(* Logix 5000 project; controller QW361 vendor 1 type 14 code 107 rev 32.11; software revision 32.00; part 17 of 20 *)

        [64].log_data[1].valid := 1, [64].log_data[2].time := 3599.999, [64].log_data[2].valid := 1, [64].log_data[3].time := 3599.999, [64].log_data[3].valid := 1, [64].log_data[4].min := 0.48812497, [64].log_data[4].max := 1.0068749, [64].log_data[4].total := 2935.025, [64].log_data[4].time := 3599.999, [64].log_data[4].minminute := 43, [64].log_data[4].maxminute := 34, [64].log_data[4].valid := 1, [64].log_data[5].max := 7.16125, [64].log_data[5].total := 3457.7583, [64].log_data[5].time := 3599.999, [64].log_data[5].maxminute := 35, [64].log_data[5].valid := 1, [64].log_data[6].valid := 1, [64].log_data[7].valid := 1, [64].log_data[8].valid := 1, [64].log_data[9].valid := 1, [64].log_data[10].valid := 1, [64].log_data[11].valid := 1, [64].log_data[12].valid := 1, [64].log_data[13].valid := 1, [64].log_data[14].valid := 1, [64].log_data[15].valid := 1, [64].log_data[16].valid := 1, [64].log_data[17].valid := 1, [64].log_data[18].valid := 1, [64].log_data[19].valid := 1, [64].time.Year := 2022, [64].time.Month := 4, [64].time.Day := 29, [64].time.Hour := 9, [64].time.Minute := 59, [64].time.Second := 59, [64].time.DST_ON := 1, [65].log_data[0].min := 1.0, [65].log_data[0].max := 1.0, [65].log_data[0].total := 3600.001, [65].log_data[0].time := 3600.001, [65].log_data[0].valid := 1, [65].log_data[1].time := 3600.001, [65].log_data[1].valid := 1, [65].log_data[2].max := 1.0, [65].log_data[2].total := 261.25, [65].log_data[2].time := 3600.001, [65].log_data[2].maxminute := 55, [65].log_data[2].valid := 1, [65].log_data[3].time := 3600.001, [65].log_data[3].valid := 1, [65].log_data[4].min := 0.64125, [65].log_data[4].max := 1.00875, [65].log_data[4].total := 3102.0618, [65].log_data[4].time := 3600.001, [65].log_data[4].maxminute := 55, [65].log_data[4].valid := 1, [65].log_data[5].max := 7.21375, [65].log_data[5].total := 1816.54,
        [65].log_data[5].time := 3600.001, [65].log_data[5].maxminute := 56, [65].log_data[5].valid := 1, [65].log_data[6].valid := 1, [65].log_data[7].valid := 1, [65].log_data[8].valid := 1, [65].log_data[9].valid := 1, [65].log_data[10].valid := 1, [65].log_data[11].valid := 1, [65].log_data[12].valid := 1, [65].log_data[13].valid := 1, [65].log_data[14].valid := 1, [65].log_data[15].valid := 1, [65].log_data[16].valid := 1, [65].log_data[17].valid := 1, [65].log_data[18].valid := 1, [65].log_data[19].valid := 1, [65].time.Year := 2022, [65].time.Month := 4, [65].time.Day := 29, [65].time.Hour := 10, [65].time.Minute := 59, [65].time.Second := 59, [65].time.DST_ON := 1, [66].log_data[0].min := 1.0, [66].log_data[0].max := 1.0, [66].log_data[0].total := 3600.0, [66].log_data[0].time := 3600.0, [66].log_data[0].valid := 1, [66].log_data[1].time := 3600.0, [66].log_data[1].valid := 1, [66].log_data[2].max := 1.0, [66].log_data[2].total := 236.25, [66].log_data[2].time := 3600.0, [66].log_data[2].minminute := 3, [66].log_data[2].valid := 1, [66].log_data[3].time := 3600.0, [66].log_data[3].valid := 1, [66].log_data[4].min := 0.48812497, [66].log_data[4].max := 0.93375, [66].log_data[4].total := 2553.6604, [66].log_data[4].time := 3600.0, [66].log_data[4].minminute := 4, [66].log_data[4].maxminute := 58, [66].log_data[4].valid := 1, [66].log_data[5].max := 7.1512504, [66].log_data[5].total := 1708.433, [66].log_data[5].time := 3600.0, [66].log_data[5].minminute := 4, [66].log_data[5].maxminute := 1, [66].log_data[5].valid := 1, [66].log_data[6].valid := 1, [66].log_data[7].valid := 1, [66].log_data[8].valid := 1, [66].log_data[9].valid := 1, [66].log_data[10].valid := 1, [66].log_data[11].valid := 1, [66].log_data[12].valid := 1, [66].log_data[13].valid := 1, [66].log_data[14].valid := 1,
        [66].log_data[15].valid := 1, [66].log_data[16].valid := 1, [66].log_data[17].valid := 1, [66].log_data[18].valid := 1, [66].log_data[19].valid := 1, [66].time.Year := 2022, [66].time.Month := 4, [66].time.Day := 29, [66].time.Hour := 11, [66].time.Minute := 59, [66].time.Second := 59, [66].time.DST_ON := 1, [67].log_data[0].min := 1.0, [67].log_data[0].max := 1.0, [67].log_data[0].total := 3600.0, [67].log_data[0].time := 3600.0, [67].log_data[0].valid := 1, [67].log_data[1].max := 1.0, [67].log_data[1].total := 497.5, [67].log_data[1].time := 3600.0, [67].log_data[1].maxminute := 16, [67].log_data[1].valid := 1, [67].log_data[2].time := 3600.0, [67].log_data[2].valid := 1, [67].log_data[3].time := 3600.0, [67].log_data[3].valid := 1, [67].log_data[4].min := 0.48812497, [67].log_data[4].max := 1.0024999, [67].log_data[4].total := 2646.7375, [67].log_data[4].time := 3600.0, [67].log_data[4].minminute := 24, [67].log_data[4].maxminute := 16, [67].log_data[4].valid := 1, [67].log_data[5].max := 7.1425004, [67].log_data[5].total := 3489.1882, [67].log_data[5].time := 3600.0, [67].log_data[5].maxminute := 17, [67].log_data[5].valid := 1, [67].log_data[6].valid := 1, [67].log_data[7].valid := 1, [67].log_data[8].valid := 1, [67].log_data[9].valid := 1, [67].log_data[10].valid := 1, [67].log_data[11].valid := 1, [67].log_data[12].valid := 1, [67].log_data[13].valid := 1, [67].log_data[14].valid := 1, [67].log_data[15].valid := 1, [67].log_data[16].valid := 1, [67].log_data[17].valid := 1, [67].log_data[18].valid := 1, [67].log_data[19].valid := 1, [67].time.Year := 2022, [67].time.Month := 4, [67].time.Day := 29, [67].time.Hour := 12, [67].time.Minute := 59, [67].time.Second := 59, [67].time.DST_ON := 1, [68].log_data[0].min := 1.0,
        [68].log_data[0].max := 1.0, [68].log_data[0].total := 3600.001, [68].log_data[0].time := 3600.001, [68].log_data[0].valid := 1, [68].log_data[1].time := 3600.001, [68].log_data[1].valid := 1, [68].log_data[2].time := 3600.001, [68].log_data[2].valid := 1, [68].log_data[3].time := 3600.001, [68].log_data[3].valid := 1, [68].log_data[4].min := 0.71812505, [68].log_data[4].max := 0.94875, [68].log_data[4].total := 3074.6538, [68].log_data[4].time := 3600.001, [68].log_data[4].maxminute := 56, [68].log_data[4].valid := 1, [68].log_data[5].time := 3600.001, [68].log_data[5].valid := 1, [68].log_data[6].valid := 1, [68].log_data[7].valid := 1, [68].log_data[8].valid := 1, [68].log_data[9].valid := 1, [68].log_data[10].valid := 1, [68].log_data[11].valid := 1, [68].log_data[12].valid := 1, [68].log_data[13].valid := 1, [68].log_data[14].valid := 1, [68].log_data[15].valid := 1, [68].log_data[16].valid := 1, [68].log_data[17].valid := 1, [68].log_data[18].valid := 1, [68].log_data[19].valid := 1, [68].time.Year := 2022, [68].time.Month := 4, [68].time.Day := 29, [68].time.Hour := 13, [68].time.Minute := 59, [68].time.Second := 59, [68].time.DST_ON := 1, [69].log_data[0].min := 1.0, [69].log_data[0].max := 1.0, [69].log_data[0].total := 3599.999, [69].log_data[0].time := 3599.999, [69].log_data[0].valid := 1, [69].log_data[1].time := 3599.999, [69].log_data[1].valid := 1, [69].log_data[2].max := 1.0, [69].log_data[2].total := 480.5, [69].log_data[2].time := 3599.999, [69].log_data[2].maxminute := 26, [69].log_data[2].valid := 1, [69].log_data[3].time := 3599.999, [69].log_data[3].valid := 1, [69].log_data[4].min := 0.48749998, [69].log_data[4].max := 1.0068749, [69].log_data[4].total := 2784.5537, [69].log_data[4].time := 3599.999, [69].log_data[4].minminute := 34, [69].log_data[4].maxminute := 26, [69].log_data[4].valid := 1,
        [69].log_data[5].max := 7.2375, [69].log_data[5].total := 3409.78, [69].log_data[5].time := 3599.999, [69].log_data[5].maxminute := 26, [69].log_data[5].valid := 1, [69].log_data[6].valid := 1, [69].log_data[7].valid := 1, [69].log_data[8].valid := 1, [69].log_data[9].valid := 1, [69].log_data[10].valid := 1, [69].log_data[11].valid := 1, [69].log_data[12].valid := 1, [69].log_data[13].valid := 1, [69].log_data[14].valid := 1, [69].log_data[15].valid := 1, [69].log_data[16].valid := 1, [69].log_data[17].valid := 1, [69].log_data[18].valid := 1, [69].log_data[19].valid := 1, [69].time.Year := 2022, [69].time.Month := 4, [69].time.Day := 29, [69].time.Hour := 14, [69].time.Minute := 59, [69].time.Second := 59, [69].time.DST_ON := 1, [70].log_data[0].min := 1.0, [70].log_data[0].max := 1.0, [70].log_data[0].total := 3600.001, [70].log_data[0].time := 3600.001, [70].log_data[0].valid := 1, [70].log_data[1].time := 3600.001, [70].log_data[1].valid := 1, [70].log_data[2].time := 3600.001, [70].log_data[2].valid := 1, [70].log_data[3].time := 3600.001, [70].log_data[3].valid := 1, [70].log_data[4].min := 0.64187497, [70].log_data[4].max := 0.91875005, [70].log_data[4].total := 2832.5027, [70].log_data[4].time := 3600.001, [70].log_data[4].maxminute := 56, [70].log_data[4].valid := 1, [70].log_data[5].time := 3600.001, [70].log_data[5].valid := 1, [70].log_data[6].valid := 1, [70].log_data[7].valid := 1, [70].log_data[8].valid := 1, [70].log_data[9].valid := 1, [70].log_data[10].valid := 1, [70].log_data[11].valid := 1, [70].log_data[12].valid := 1, [70].log_data[13].valid := 1, [70].log_data[14].valid := 1, [70].log_data[15].valid := 1, [70].log_data[16].valid := 1, [70].log_data[17].valid := 1, [70].log_data[18].valid := 1, [70].log_data[19].valid := 1, [70].time.Year := 2022,
        [70].time.Month := 4, [70].time.Day := 29, [70].time.Hour := 15, [70].time.Minute := 59, [70].time.Second := 59, [70].time.DST_ON := 1, [71].log_data[0].min := 1.0, [71].log_data[0].max := 1.0, [71].log_data[0].total := 3600.0, [71].log_data[0].time := 3600.0, [71].log_data[0].valid := 1, [71].log_data[1].max := 1.0, [71].log_data[1].total := 486.0, [71].log_data[1].time := 3600.0, [71].log_data[1].maxminute := 33, [71].log_data[1].valid := 1, [71].log_data[2].time := 3600.0, [71].log_data[2].valid := 1, [71].log_data[3].time := 3600.0, [71].log_data[3].valid := 1, [71].log_data[4].min := 0.48749998, [71].log_data[4].max := 1.00375, [71].log_data[4].total := 2909.2458, [71].log_data[4].time := 3600.0, [71].log_data[4].minminute := 41, [71].log_data[4].maxminute := 33, [71].log_data[4].valid := 1, [71].log_data[5].max := 7.1525, [71].log_data[5].total := 3410.604, [71].log_data[5].time := 3600.0, [71].log_data[5].maxminute := 34, [71].log_data[5].valid := 1, [71].log_data[6].valid := 1, [71].log_data[7].valid := 1, [71].log_data[8].valid := 1, [71].log_data[9].valid := 1, [71].log_data[10].valid := 1, [71].log_data[11].valid := 1, [71].log_data[12].valid := 1, [71].log_data[13].valid := 1, [71].log_data[14].valid := 1, [71].log_data[15].valid := 1, [71].log_data[16].valid := 1, [71].log_data[17].valid := 1, [71].log_data[18].valid := 1, [71].log_data[19].valid := 1, [71].time.Year := 2022, [71].time.Month := 4, [71].time.Day := 29, [71].time.Hour := 16, [71].time.Minute := 59, [71].time.Second := 59, [71].time.DST_ON := 1, [72].log_data[0].min := 1.0, [72].log_data[0].max := 1.0, [72].log_data[0].total := 3599.999, [72].log_data[0].time := 3599.999, [72].log_data[0].valid := 1, [72].log_data[1].time := 3599.999, [72].log_data[1].valid := 1,
        [72].log_data[2].time := 3599.999, [72].log_data[2].valid := 1, [72].log_data[3].time := 3599.999, [72].log_data[3].valid := 1, [72].log_data[4].min := 0.57937497, [72].log_data[4].max := 0.8725, [72].log_data[4].total := 2595.1763, [72].log_data[4].time := 3599.999, [72].log_data[4].maxminute := 59, [72].log_data[4].valid := 1, [72].log_data[5].time := 3599.999, [72].log_data[5].valid := 1, [72].log_data[6].valid := 1, [72].log_data[7].valid := 1, [72].log_data[8].valid := 1, [72].log_data[9].valid := 1, [72].log_data[10].valid := 1, [72].log_data[11].valid := 1, [72].log_data[12].valid := 1, [72].log_data[13].valid := 1, [72].log_data[14].valid := 1, [72].log_data[15].valid := 1, [72].log_data[16].valid := 1, [72].log_data[17].valid := 1, [72].log_data[18].valid := 1, [72].log_data[19].valid := 1, [72].time.Year := 2022, [72].time.Month := 4, [72].time.Day := 29, [72].time.Hour := 17, [72].time.Minute := 59, [72].time.Second := 59, [72].time.DST_ON := 1, [73].log_data[0].min := 1.0, [73].log_data[0].max := 1.0, [73].log_data[0].total := 3600.0, [73].log_data[0].time := 3600.0, [73].log_data[0].valid := 1, [73].log_data[1].time := 3600.0, [73].log_data[1].valid := 1, [73].log_data[2].max := 1.0, [73].log_data[2].total := 486.0, [73].log_data[2].time := 3600.0, [73].log_data[2].maxminute := 50, [73].log_data[2].valid := 1, [73].log_data[3].time := 3600.0, [73].log_data[3].valid := 1, [73].log_data[4].min := 0.48749998, [73].log_data[4].max := 1.00625, [73].log_data[4].total := 3274.2031, [73].log_data[4].time := 3600.0, [73].log_data[4].minminute := 58, [73].log_data[4].maxminute := 50, [73].log_data[4].valid := 1, [73].log_data[5].max := 7.235, [73].log_data[5].total := 3447.0845, [73].log_data[5].time := 3600.0, [73].log_data[5].maxminute := 51, [73].log_data[5].valid := 1, [73].log_data[6].valid := 1,
        [73].log_data[7].valid := 1, [73].log_data[8].valid := 1, [73].log_data[9].valid := 1, [73].log_data[10].valid := 1, [73].log_data[11].valid := 1, [73].log_data[12].valid := 1, [73].log_data[13].valid := 1, [73].log_data[14].valid := 1, [73].log_data[15].valid := 1, [73].log_data[16].valid := 1, [73].log_data[17].valid := 1, [73].log_data[18].valid := 1, [73].log_data[19].valid := 1, [73].time.Year := 2022, [73].time.Month := 4, [73].time.Day := 29, [73].time.Hour := 18, [73].time.Minute := 59, [73].time.Second := 59, [73].time.DST_ON := 1, [74].log_data[0].min := 1.0, [74].log_data[0].max := 1.0, [74].log_data[0].total := 3600.0, [74].log_data[0].time := 3600.0, [74].log_data[0].valid := 1, [74].log_data[1].time := 3600.0, [74].log_data[1].valid := 1, [74].log_data[2].time := 3600.0, [74].log_data[2].valid := 1, [74].log_data[3].time := 3600.0, [74].log_data[3].valid := 1, [74].log_data[4].min := 0.48749998, [74].log_data[4].max := 0.9024999, [74].log_data[4].total := 2510.1887, [74].log_data[4].time := 3600.0, [74].log_data[4].maxminute := 57, [74].log_data[4].valid := 1, [74].log_data[5].time := 3600.0, [74].log_data[5].valid := 1, [74].log_data[6].valid := 1, [74].log_data[7].valid := 1, [74].log_data[8].valid := 1, [74].log_data[9].valid := 1, [74].log_data[10].valid := 1, [74].log_data[11].valid := 1, [74].log_data[12].valid := 1, [74].log_data[13].valid := 1, [74].log_data[14].valid := 1, [74].log_data[15].valid := 1, [74].log_data[16].valid := 1, [74].log_data[17].valid := 1, [74].log_data[18].valid := 1, [74].log_data[19].valid := 1, [74].time.Year := 2022, [74].time.Month := 4, [74].time.Day := 29, [74].time.Hour := 19, [74].time.Minute := 59, [74].time.Second := 59, [74].time.DST_ON := 1,
        [75].log_data[0].min := 1.0, [75].log_data[0].max := 1.0, [75].log_data[0].total := 3599.999, [75].log_data[0].time := 3599.999, [75].log_data[0].valid := 1, [75].log_data[1].max := 1.0, [75].log_data[1].total := 512.0, [75].log_data[1].time := 3599.999, [75].log_data[1].maxminute := 25, [75].log_data[1].valid := 1, [75].log_data[2].time := 3599.999, [75].log_data[2].valid := 1, [75].log_data[3].time := 3599.999, [75].log_data[3].valid := 1, [75].log_data[4].min := 0.48749998, [75].log_data[4].max := 1.00875, [75].log_data[4].total := 2836.993, [75].log_data[4].time := 3599.999, [75].log_data[4].minminute := 34, [75].log_data[4].maxminute := 25, [75].log_data[4].valid := 1, [75].log_data[5].max := 7.1650004, [75].log_data[5].total := 3593.2307, [75].log_data[5].time := 3599.999, [75].log_data[5].maxminute := 26, [75].log_data[5].valid := 1, [75].log_data[6].valid := 1, [75].log_data[7].valid := 1, [75].log_data[8].valid := 1, [75].log_data[9].valid := 1, [75].log_data[10].valid := 1, [75].log_data[11].valid := 1, [75].log_data[12].valid := 1, [75].log_data[13].valid := 1, [75].log_data[14].valid := 1, [75].log_data[15].valid := 1, [75].log_data[16].valid := 1, [75].log_data[17].valid := 1, [75].log_data[18].valid := 1, [75].log_data[19].valid := 1, [75].time.Year := 2022, [75].time.Month := 4, [75].time.Day := 29, [75].time.Hour := 20, [75].time.Minute := 59, [75].time.Second := 59, [75].time.DST_ON := 1, [76].log_data[0].min := 1.0, [76].log_data[0].max := 1.0, [76].log_data[0].total := 3600.0, [76].log_data[0].time := 3600.0, [76].log_data[0].valid := 1, [76].log_data[1].time := 3600.0, [76].log_data[1].valid := 1, [76].log_data[2].max := 1.0, [76].log_data[2].total := 493.0, [76].log_data[2].time := 3600.0, [76].log_data[2].maxminute := 50, [76].log_data[2].valid := 1, [76].log_data[3].time := 3600.0,
        [76].log_data[3].valid := 1, [76].log_data[4].min := 0.48812497, [76].log_data[4].max := 1.005, [76].log_data[4].total := 3163.5645, [76].log_data[4].time := 3600.0, [76].log_data[4].minminute := 58, [76].log_data[4].maxminute := 50, [76].log_data[4].valid := 1, [76].log_data[5].max := 7.24375, [76].log_data[5].total := 3493.379, [76].log_data[5].time := 3600.0, [76].log_data[5].maxminute := 50, [76].log_data[5].valid := 1, [76].log_data[6].valid := 1, [76].log_data[7].valid := 1, [76].log_data[8].valid := 1, [76].log_data[9].valid := 1, [76].log_data[10].valid := 1, [76].log_data[11].valid := 1, [76].log_data[12].valid := 1, [76].log_data[13].valid := 1, [76].log_data[14].valid := 1, [76].log_data[15].valid := 1, [76].log_data[16].valid := 1, [76].log_data[17].valid := 1, [76].log_data[18].valid := 1, [76].log_data[19].valid := 1, [76].time.Year := 2022, [76].time.Month := 4, [76].time.Day := 29, [76].time.Hour := 21, [76].time.Minute := 59, [76].time.Second := 59, [76].time.DST_ON := 1, [77].log_data[0].min := 1.0, [77].log_data[0].max := 1.0, [77].log_data[0].total := 3600.0, [77].log_data[0].time := 3600.0, [77].log_data[0].valid := 1, [77].log_data[1].time := 3600.0, [77].log_data[1].valid := 1, [77].log_data[2].time := 3600.0, [77].log_data[2].valid := 1, [77].log_data[3].time := 3600.0, [77].log_data[3].valid := 1, [77].log_data[4].min := 0.5025, [77].log_data[4].max := 0.94875, [77].log_data[4].total := 2784.093, [77].log_data[4].time := 3600.0, [77].log_data[4].maxminute := 57, [77].log_data[4].valid := 1, [77].log_data[5].max := 0.0025000002, [77].log_data[5].total := 0.59032303, [77].log_data[5].time := 3600.0, [77].log_data[5].maxminute := 54, [77].log_data[5].valid := 1, [77].log_data[6].valid := 1, [77].log_data[7].valid := 1, [77].log_data[8].valid := 1, [77].log_data[9].valid := 1,
        [77].log_data[10].valid := 1, [77].log_data[11].valid := 1, [77].log_data[12].valid := 1, [77].log_data[13].valid := 1, [77].log_data[14].valid := 1, [77].log_data[15].valid := 1, [77].log_data[16].valid := 1, [77].log_data[17].valid := 1, [77].log_data[18].valid := 1, [77].log_data[19].valid := 1, [77].time.Year := 2022, [77].time.Month := 4, [77].time.Day := 29, [77].time.Hour := 22, [77].time.Minute := 59, [77].time.Second := 59, [77].time.DST_ON := 1, [78].log_data[0].min := 1.0, [78].log_data[0].max := 1.0, [78].log_data[0].total := 3600.0, [78].log_data[0].time := 3600.0, [78].log_data[0].valid := 1, [78].log_data[1].max := 1.0, [78].log_data[1].total := 483.5, [78].log_data[1].time := 3600.0, [78].log_data[1].maxminute := 24, [78].log_data[1].valid := 1, [78].log_data[2].time := 3600.0, [78].log_data[2].valid := 1, [78].log_data[3].time := 3600.0, [78].log_data[3].valid := 1, [78].log_data[4].min := 0.48812497, [78].log_data[4].max := 1.0068749, [78].log_data[4].total := 2779.4797, [78].log_data[4].time := 3600.0, [78].log_data[4].minminute := 32, [78].log_data[4].maxminute := 24, [78].log_data[4].valid := 1, [78].log_data[5].max := 7.13875, [78].log_data[5].total := 3404.901, [78].log_data[5].time := 3600.0, [78].log_data[5].maxminute := 25, [78].log_data[5].valid := 1, [78].log_data[6].valid := 1, [78].log_data[7].valid := 1, [78].log_data[8].valid := 1, [78].log_data[9].valid := 1, [78].log_data[10].valid := 1, [78].log_data[11].valid := 1, [78].log_data[12].valid := 1, [78].log_data[13].valid := 1, [78].log_data[14].valid := 1, [78].log_data[15].valid := 1, [78].log_data[16].valid := 1, [78].log_data[17].valid := 1, [78].log_data[18].valid := 1, [78].log_data[19].valid := 1, [78].time.Year := 2022, [78].time.Month := 4, [78].time.Day := 29,
        [78].time.Hour := 23, [78].time.Minute := 59, [78].time.Second := 59, [78].time.DST_ON := 1, [79].log_data[0].min := 1.0, [79].log_data[0].max := 1.0, [79].log_data[0].total := 3600.0, [79].log_data[0].time := 3600.0, [79].log_data[0].valid := 1, [79].log_data[1].time := 3600.0, [79].log_data[1].valid := 1, [79].log_data[2].time := 3600.0, [79].log_data[2].valid := 1, [79].log_data[3].time := 3600.0, [79].log_data[3].valid := 1, [79].log_data[4].min := 0.71812505, [79].log_data[4].max := 0.98, [79].log_data[4].total := 3211.9824, [79].log_data[4].time := 3600.0, [79].log_data[4].maxminute := 53, [79].log_data[4].valid := 1, [79].log_data[5].max := 0.0012500001, [79].log_data[5].total := 1.0756322, [79].log_data[5].time := 3600.0, [79].log_data[5].valid := 1, [79].log_data[6].valid := 1, [79].log_data[7].valid := 1, [79].log_data[8].valid := 1, [79].log_data[9].valid := 1, [79].log_data[10].valid := 1, [79].log_data[11].valid := 1, [79].log_data[12].valid := 1, [79].log_data[13].valid := 1, [79].log_data[14].valid := 1, [79].log_data[15].valid := 1, [79].log_data[16].valid := 1, [79].log_data[17].valid := 1, [79].log_data[18].valid := 1, [79].log_data[19].valid := 1, [79].time.Year := 2022, [79].time.Month := 4, [79].time.Day := 30, [79].time.Minute := 59, [79].time.Second := 59, [79].time.DST_ON := 1, [80].log_data[0].min := 1.0, [80].log_data[0].max := 1.0, [80].log_data[0].total := 3600.0, [80].log_data[0].time := 3600.0, [80].log_data[0].valid := 1, [80].log_data[1].time := 3600.0, [80].log_data[1].valid := 1, [80].log_data[2].max := 1.0, [80].log_data[2].total := 477.0, [80].log_data[2].time := 3600.0, [80].log_data[2].maxminute := 10, [80].log_data[2].valid := 1, [80].log_data[3].time := 3600.0, [80].log_data[3].valid := 1, [80].log_data[4].min := 0.48812497,
        [80].log_data[4].max := 1.0068749, [80].log_data[4].total := 2421.8188, [80].log_data[4].time := 3600.0, [80].log_data[4].minminute := 18, [80].log_data[4].maxminute := 10, [80].log_data[4].valid := 1, [80].log_data[5].max := 7.2237496, [80].log_data[5].total := 3382.9375, [80].log_data[5].time := 3600.0, [80].log_data[5].maxminute := 11, [80].log_data[5].valid := 1, [80].log_data[6].valid := 1, [80].log_data[7].valid := 1, [80].log_data[8].valid := 1, [80].log_data[9].valid := 1, [80].log_data[10].valid := 1, [80].log_data[11].valid := 1, [80].log_data[12].valid := 1, [80].log_data[13].valid := 1, [80].log_data[14].valid := 1, [80].log_data[15].valid := 1, [80].log_data[16].valid := 1, [80].log_data[17].valid := 1, [80].log_data[18].valid := 1, [80].log_data[19].valid := 1, [80].time.Year := 2022, [80].time.Month := 4, [80].time.Day := 30, [80].time.Hour := 1, [80].time.Minute := 59, [80].time.Second := 59, [80].time.DST_ON := 1, [81].log_data[0].min := 1.0, [81].log_data[0].max := 1.0, [81].log_data[0].total := 3600.0, [81].log_data[0].time := 3600.0, [81].log_data[0].valid := 1, [81].log_data[1].time := 3600.0, [81].log_data[1].valid := 1, [81].log_data[2].time := 3600.0, [81].log_data[2].valid := 1, [81].log_data[3].time := 3600.0, [81].log_data[3].valid := 1, [81].log_data[4].min := 0.656875, [81].log_data[4].max := 0.8268749, [81].log_data[4].total := 2698.259, [81].log_data[4].time := 3600.0, [81].log_data[4].maxminute := 55, [81].log_data[4].valid := 1, [81].log_data[5].max := 0.0012500001, [81].log_data[5].total := 2.276786, [81].log_data[5].time := 3600.0, [81].log_data[5].valid := 1, [81].log_data[6].valid := 1, [81].log_data[7].valid := 1, [81].log_data[8].valid := 1, [81].log_data[9].valid := 1, [81].log_data[10].valid := 1, [81].log_data[11].valid := 1, [81].log_data[12].valid := 1,
        [81].log_data[13].valid := 1, [81].log_data[14].valid := 1, [81].log_data[15].valid := 1, [81].log_data[16].valid := 1, [81].log_data[17].valid := 1, [81].log_data[18].valid := 1, [81].log_data[19].valid := 1, [81].time.Year := 2022, [81].time.Month := 4, [81].time.Day := 30, [81].time.Hour := 2, [81].time.Minute := 59, [81].time.Second := 59, [81].time.DST_ON := 1, [82].log_data[0].min := 1.0, [82].log_data[0].max := 1.0, [82].log_data[0].total := 3600.0, [82].log_data[0].time := 3600.0, [82].log_data[0].valid := 1, [82].log_data[1].time := 3600.0, [82].log_data[1].valid := 1, [82].log_data[2].time := 3600.0, [82].log_data[2].valid := 1, [82].log_data[3].time := 3600.0, [82].log_data[3].valid := 1, [82].log_data[4].min := 0.82625, [82].log_data[4].max := 0.91875005, [82].log_data[4].total := 3186.939, [82].log_data[4].time := 3600.0, [82].log_data[4].maxminute := 48, [82].log_data[4].valid := 1, [82].log_data[5].max := 0.0012500001, [82].log_data[5].total := 2.8984814, [82].log_data[5].time := 3600.0, [82].log_data[5].valid := 1, [82].log_data[6].valid := 1, [82].log_data[7].valid := 1, [82].log_data[8].valid := 1, [82].log_data[9].valid := 1, [82].log_data[10].valid := 1, [82].log_data[11].valid := 1, [82].log_data[12].valid := 1, [82].log_data[13].valid := 1, [82].log_data[14].valid := 1, [82].log_data[15].valid := 1, [82].log_data[16].valid := 1, [82].log_data[17].valid := 1, [82].log_data[18].valid := 1, [82].log_data[19].valid := 1, [82].time.Year := 2022, [82].time.Month := 4, [82].time.Day := 30, [82].time.Hour := 3, [82].time.Minute := 59, [82].time.Second := 59, [82].time.DST_ON := 1, [83].log_data[0].min := 1.0, [83].log_data[0].max := 1.0, [83].log_data[0].total := 3600.0, [83].log_data[0].time := 3600.0,
        [83].log_data[0].valid := 1, [83].log_data[1].time := 3600.0, [83].log_data[1].valid := 1, [83].log_data[2].time := 3600.0, [83].log_data[2].valid := 1, [83].log_data[3].time := 3600.0, [83].log_data[3].valid := 1, [83].log_data[4].min := 0.91875005, [83].log_data[4].max := 0.9650001, [83].log_data[4].total := 3411.9158, [83].log_data[4].time := 3600.0, [83].log_data[4].maxminute := 42, [83].log_data[4].valid := 1, [83].log_data[5].max := 0.0012500001, [83].log_data[5].total := 2.8228402, [83].log_data[5].time := 3600.0, [83].log_data[5].valid := 1, [83].log_data[6].valid := 1, [83].log_data[7].valid := 1, [83].log_data[8].valid := 1, [83].log_data[9].valid := 1, [83].log_data[10].valid := 1, [83].log_data[11].valid := 1, [83].log_data[12].valid := 1, [83].log_data[13].valid := 1, [83].log_data[14].valid := 1, [83].log_data[15].valid := 1, [83].log_data[16].valid := 1, [83].log_data[17].valid := 1, [83].log_data[18].valid := 1, [83].log_data[19].valid := 1, [83].time.Year := 2022, [83].time.Month := 4, [83].time.Day := 30, [83].time.Hour := 4, [83].time.Minute := 59, [83].time.Second := 59, [83].time.DST_ON := 1, [84].log_data[0].min := 1.0, [84].log_data[0].max := 1.0, [84].log_data[0].total := 3599.999, [84].log_data[0].time := 3599.999, [84].log_data[0].valid := 1, [84].log_data[1].max := 1.0, [84].log_data[1].total := 154.75, [84].log_data[1].time := 3599.999, [84].log_data[1].maxminute := 57, [84].log_data[1].valid := 1, [84].log_data[2].time := 3599.999, [84].log_data[2].valid := 1, [84].log_data[3].time := 3599.999, [84].log_data[3].valid := 1, [84].log_data[4].min := 0.9125, [84].log_data[4].max := 1.00125, [84].log_data[4].total := 3550.91, [84].log_data[4].time := 3599.999, [84].log_data[4].minminute := 59, [84].log_data[4].maxminute := 57, [84].log_data[4].valid := 1, [84].log_data[5].max := 7.1625,
        [84].log_data[5].total := 1047.2858, [84].log_data[5].time := 3599.999, [84].log_data[5].maxminute := 58, [84].log_data[5].valid := 1, [84].log_data[6].valid := 1, [84].log_data[7].valid := 1, [84].log_data[8].valid := 1, [84].log_data[9].valid := 1, [84].log_data[10].valid := 1, [84].log_data[11].valid := 1, [84].log_data[12].valid := 1, [84].log_data[13].valid := 1, [84].log_data[14].valid := 1, [84].log_data[15].valid := 1, [84].log_data[16].valid := 1, [84].log_data[17].valid := 1, [84].log_data[18].valid := 1, [84].log_data[19].valid := 1, [84].time.Year := 2022, [84].time.Month := 4, [84].time.Day := 30, [84].time.Hour := 5, [84].time.Minute := 59, [84].time.Second := 59, [84].time.DST_ON := 1, [85].log_data[0].min := 1.0, [85].log_data[0].max := 1.0, [85].log_data[0].total := 3600.0, [85].log_data[0].time := 3600.0, [85].log_data[0].valid := 1, [85].log_data[1].max := 1.0, [85].log_data[1].total := 317.25, [85].log_data[1].time := 3600.0, [85].log_data[1].minminute := 5, [85].log_data[1].valid := 1, [85].log_data[2].time := 3600.0, [85].log_data[2].valid := 1, [85].log_data[3].time := 3600.0, [85].log_data[3].valid := 1, [85].log_data[4].min := 0.48812497, [85].log_data[4].max := 0.9125, [85].log_data[4].total := 1935.4558, [85].log_data[4].time := 3600.0, [85].log_data[4].minminute := 5, [85].log_data[4].valid := 1, [85].log_data[5].max := 7.1225, [85].log_data[5].total := 2269.2898, [85].log_data[5].time := 3600.0, [85].log_data[5].minminute := 5, [85].log_data[5].valid := 1, [85].log_data[6].valid := 1, [85].log_data[7].valid := 1, [85].log_data[8].valid := 1, [85].log_data[9].valid := 1, [85].log_data[10].valid := 1, [85].log_data[11].valid := 1, [85].log_data[12].valid := 1, [85].log_data[13].valid := 1, [85].log_data[14].valid := 1, [85].log_data[15].valid := 1,
        [85].log_data[16].valid := 1, [85].log_data[17].valid := 1, [85].log_data[18].valid := 1, [85].log_data[19].valid := 1, [85].time.Year := 2022, [85].time.Month := 4, [85].time.Day := 30, [85].time.Hour := 6, [85].time.Minute := 59, [85].time.Second := 59, [85].time.DST_ON := 1, [86].log_data[0].min := 1.0, [86].log_data[0].max := 1.0, [86].log_data[0].total := 3600.0, [86].log_data[0].time := 3600.0, [86].log_data[0].valid := 1, [86].log_data[1].time := 3600.0, [86].log_data[1].valid := 1, [86].log_data[2].time := 3600.0, [86].log_data[2].valid := 1, [86].log_data[3].time := 3600.0, [86].log_data[3].valid := 1, [86].log_data[4].min := 0.56500006, [86].log_data[4].max := 0.70375, [86].log_data[4].total := 2291.6409, [86].log_data[4].time := 3600.0, [86].log_data[4].maxminute := 55, [86].log_data[4].valid := 1, [86].log_data[5].max := 0.0025000002, [86].log_data[5].total := 1.7577057, [86].log_data[5].time := 3600.0, [86].log_data[5].maxminute := 35, [86].log_data[5].valid := 1, [86].log_data[6].valid := 1, [86].log_data[7].valid := 1, [86].log_data[8].valid := 1, [86].log_data[9].valid := 1, [86].log_data[10].valid := 1, [86].log_data[11].valid := 1, [86].log_data[12].valid := 1, [86].log_data[13].valid := 1, [86].log_data[14].valid := 1, [86].log_data[15].valid := 1, [86].log_data[16].valid := 1, [86].log_data[17].valid := 1, [86].log_data[18].valid := 1, [86].log_data[19].valid := 1, [86].time.Year := 2022, [86].time.Month := 4, [86].time.Day := 30, [86].time.Hour := 7, [86].time.Minute := 59, [86].time.Second := 59, [86].time.DST_ON := 1, [87].log_data[0].min := 1.0, [87].log_data[0].max := 1.0, [87].log_data[0].total := 3599.999, [87].log_data[0].time := 3599.999, [87].log_data[0].valid := 1, [87].log_data[1].time := 3599.999,
        [87].log_data[1].valid := 1, [87].log_data[2].time := 3599.999, [87].log_data[2].valid := 1, [87].log_data[3].time := 3599.999, [87].log_data[3].valid := 1, [87].log_data[4].min := 0.703125, [87].log_data[4].max := 0.9024999, [87].log_data[4].total := 2915.0146, [87].log_data[4].time := 3599.999, [87].log_data[4].maxminute := 55, [87].log_data[4].valid := 1, [87].log_data[5].max := 0.0025000002, [87].log_data[5].total := 0.7278249, [87].log_data[5].time := 3599.999, [87].log_data[5].maxminute := 1, [87].log_data[5].valid := 1, [87].log_data[6].valid := 1, [87].log_data[7].valid := 1, [87].log_data[8].valid := 1, [87].log_data[9].valid := 1, [87].log_data[10].valid := 1, [87].log_data[11].valid := 1, [87].log_data[12].valid := 1, [87].log_data[13].valid := 1, [87].log_data[14].valid := 1, [87].log_data[15].valid := 1, [87].log_data[16].valid := 1, [87].log_data[17].valid := 1, [87].log_data[18].valid := 1, [87].log_data[19].valid := 1, [87].time.Year := 2022, [87].time.Month := 4, [87].time.Day := 30, [87].time.Hour := 8, [87].time.Minute := 59, [87].time.Second := 59, [87].time.DST_ON := 1, [88].log_data[0].min := 1.0, [88].log_data[0].max := 1.0, [88].log_data[0].total := 3600.0, [88].log_data[0].time := 3600.0, [88].log_data[0].valid := 1, [88].log_data[1].time := 3600.0, [88].log_data[1].valid := 1, [88].log_data[2].max := 1.0, [88].log_data[2].total := 527.0, [88].log_data[2].time := 3600.0, [88].log_data[2].maxminute := 24, [88].log_data[2].valid := 1, [88].log_data[3].time := 3600.0, [88].log_data[3].valid := 1, [88].log_data[4].min := 0.48812497, [88].log_data[4].max := 1.00875, [88].log_data[4].total := 2933.3132, [88].log_data[4].time := 3600.0, [88].log_data[4].minminute := 33, [88].log_data[4].maxminute := 24, [88].log_data[4].valid := 1, [88].log_data[5].max := 7.2199993, [88].log_data[5].total := 3743.0854,
        [88].log_data[5].time := 3600.0, [88].log_data[5].maxminute := 25, [88].log_data[5].valid := 1, [88].log_data[6].valid := 1, [88].log_data[7].valid := 1, [88].log_data[8].valid := 1, [88].log_data[9].valid := 1, [88].log_data[10].valid := 1, [88].log_data[11].valid := 1, [88].log_data[12].valid := 1, [88].log_data[13].valid := 1, [88].log_data[14].valid := 1, [88].log_data[15].valid := 1, [88].log_data[16].valid := 1, [88].log_data[17].valid := 1, [88].log_data[18].valid := 1, [88].log_data[19].valid := 1, [88].time.Year := 2022, [88].time.Month := 4, [88].time.Day := 30, [88].time.Hour := 9, [88].time.Minute := 59, [88].time.Second := 59, [88].time.DST_ON := 1, [89].log_data[0].min := 1.0, [89].log_data[0].max := 1.0, [89].log_data[0].total := 3600.0, [89].log_data[0].time := 3600.0, [89].log_data[0].valid := 1, [89].log_data[1].max := 1.0, [89].log_data[1].total := 517.5, [89].log_data[1].time := 3600.0, [89].log_data[1].maxminute := 14, [89].log_data[1].valid := 1, [89].log_data[2].time := 3600.0, [89].log_data[2].valid := 1, [89].log_data[3].time := 3600.0, [89].log_data[3].valid := 1, [89].log_data[4].min := 0.48812497, [89].log_data[4].max := 1.00875, [89].log_data[4].total := 2784.0623, [89].log_data[4].time := 3600.0, [89].log_data[4].minminute := 23, [89].log_data[4].maxminute := 14, [89].log_data[4].valid := 1, [89].log_data[5].max := 7.1687503, [89].log_data[5].total := 3641.5083, [89].log_data[5].time := 3600.0, [89].log_data[5].maxminute := 15, [89].log_data[5].valid := 1, [89].log_data[6].valid := 1, [89].log_data[7].valid := 1, [89].log_data[8].valid := 1, [89].log_data[9].valid := 1, [89].log_data[10].valid := 1, [89].log_data[11].valid := 1, [89].log_data[12].valid := 1, [89].log_data[13].valid := 1, [89].log_data[14].valid := 1, [89].log_data[15].valid := 1,
        [89].log_data[16].valid := 1, [89].log_data[17].valid := 1, [89].log_data[18].valid := 1, [89].log_data[19].valid := 1, [89].time.Year := 2022, [89].time.Month := 4, [89].time.Day := 30, [89].time.Hour := 10, [89].time.Minute := 59, [89].time.Second := 59, [89].time.DST_ON := 1, [90].log_data[0].min := 1.0, [90].log_data[0].max := 1.0, [90].log_data[0].total := 3600.001, [90].log_data[0].time := 3600.001, [90].log_data[0].valid := 1, [90].log_data[1].time := 3600.001, [90].log_data[1].valid := 1, [90].log_data[2].max := 1.0, [90].log_data[2].total := 507.0, [90].log_data[2].time := 3600.001, [90].log_data[2].maxminute := 19, [90].log_data[2].valid := 1, [90].log_data[3].time := 3600.001, [90].log_data[3].valid := 1, [90].log_data[4].min := 0.48812497, [90].log_data[4].max := 1.00875, [90].log_data[4].total := 2806.7434, [90].log_data[4].time := 3600.001, [90].log_data[4].minminute := 28, [90].log_data[4].maxminute := 20, [90].log_data[4].valid := 1, [90].log_data[5].max := 7.22875, [90].log_data[5].total := 3597.494, [90].log_data[5].time := 3600.001, [90].log_data[5].maxminute := 21, [90].log_data[5].valid := 1, [90].log_data[6].valid := 1, [90].log_data[7].valid := 1, [90].log_data[8].valid := 1, [90].log_data[9].valid := 1, [90].log_data[10].valid := 1, [90].log_data[11].valid := 1, [90].log_data[12].valid := 1, [90].log_data[13].valid := 1, [90].log_data[14].valid := 1, [90].log_data[15].valid := 1, [90].log_data[16].valid := 1, [90].log_data[17].valid := 1, [90].log_data[18].valid := 1, [90].log_data[19].valid := 1, [90].time.Year := 2022, [90].time.Month := 4, [90].time.Day := 30, [90].time.Hour := 11, [90].time.Minute := 59, [90].time.Second := 59, [90].time.DST_ON := 1, [91].log_data[0].min := 1.0, [91].log_data[0].max := 1.0,
        [91].log_data[0].total := 3599.999, [91].log_data[0].time := 3599.999, [91].log_data[0].valid := 1, [91].log_data[1].max := 1.0, [91].log_data[1].total := 503.0, [91].log_data[1].time := 3599.999, [91].log_data[1].maxminute := 31, [91].log_data[1].valid := 1, [91].log_data[2].time := 3599.999, [91].log_data[2].valid := 1, [91].log_data[3].time := 3599.999, [91].log_data[3].valid := 1, [91].log_data[4].min := 0.48812497, [91].log_data[4].max := 1.00875, [91].log_data[4].total := 2871.145, [91].log_data[4].time := 3599.999, [91].log_data[4].minminute := 40, [91].log_data[4].maxminute := 31, [91].log_data[4].valid := 1, [91].log_data[5].max := 7.15375, [91].log_data[5].total := 3531.5981, [91].log_data[5].time := 3599.999, [91].log_data[5].maxminute := 33, [91].log_data[5].valid := 1, [91].log_data[6].valid := 1, [91].log_data[7].valid := 1, [91].log_data[8].valid := 1, [91].log_data[9].valid := 1, [91].log_data[10].valid := 1, [91].log_data[11].valid := 1, [91].log_data[12].valid := 1, [91].log_data[13].valid := 1, [91].log_data[14].valid := 1, [91].log_data[15].valid := 1, [91].log_data[16].valid := 1, [91].log_data[17].valid := 1, [91].log_data[18].valid := 1, [91].log_data[19].valid := 1, [91].time.Year := 2022, [91].time.Month := 4, [91].time.Day := 30, [91].time.Hour := 12, [91].time.Minute := 59, [91].time.Second := 59, [91].time.DST_ON := 1, [92].log_data[0].min := 1.0, [92].log_data[0].max := 1.0, [92].log_data[0].total := 3600.0, [92].log_data[0].time := 3600.0, [92].log_data[0].valid := 1, [92].log_data[1].time := 3600.0, [92].log_data[1].valid := 1, [92].log_data[2].max := 1.0, [92].log_data[2].total := 495.0, [92].log_data[2].time := 3600.0, [92].log_data[2].maxminute := 49, [92].log_data[2].valid := 1, [92].log_data[3].time := 3600.0, [92].log_data[3].valid := 1, [92].log_data[4].min := 0.48749998,
        [92].log_data[4].max := 1.00875, [92].log_data[4].total := 3045.3135, [92].log_data[4].time := 3600.0, [92].log_data[4].minminute := 58, [92].log_data[4].maxminute := 49, [92].log_data[4].valid := 1, [92].log_data[5].max := 7.24625, [92].log_data[5].total := 3515.6619, [92].log_data[5].time := 3600.0, [92].log_data[5].maxminute := 51, [92].log_data[5].valid := 1, [92].log_data[6].valid := 1, [92].log_data[7].valid := 1, [92].log_data[8].valid := 1, [92].log_data[9].valid := 1, [92].log_data[10].valid := 1, [92].log_data[11].valid := 1, [92].log_data[12].valid := 1, [92].log_data[13].valid := 1, [92].log_data[14].valid := 1, [92].log_data[15].valid := 1, [92].log_data[16].valid := 1, [92].log_data[17].valid := 1, [92].log_data[18].valid := 1, [92].log_data[19].valid := 1, [92].time.Year := 2022, [92].time.Month := 4, [92].time.Day := 30, [92].time.Hour := 13, [92].time.Minute := 59, [92].time.Second := 59, [92].time.DST_ON := 1, [93].log_data[0].min := 1.0, [93].log_data[0].max := 1.0, [93].log_data[0].total := 3600.499, [93].log_data[0].time := 3600.499, [93].log_data[0].valid := 1, [93].log_data[1].time := 3600.499, [93].log_data[1].valid := 1, [93].log_data[2].time := 3600.499, [93].log_data[2].valid := 1, [93].log_data[3].time := 3600.499, [93].log_data[3].valid := 1, [93].log_data[4].min := 0.48937503, [93].log_data[4].max := 0.97937495, [93].log_data[4].total := 2772.9854, [93].log_data[4].time := 3600.499, [93].log_data[4].maxminute := 57, [93].log_data[4].valid := 1, [93].log_data[5].time := 3600.499, [93].log_data[5].valid := 1, [93].log_data[6].valid := 1, [93].log_data[7].valid := 1, [93].log_data[8].valid := 1, [93].log_data[9].valid := 1, [93].log_data[10].valid := 1, [93].log_data[11].valid := 1, [93].log_data[12].valid := 1, [93].log_data[13].valid := 1, [93].log_data[14].valid := 1,
        [93].log_data[15].valid := 1, [93].log_data[16].valid := 1, [93].log_data[17].valid := 1, [93].log_data[18].valid := 1, [93].log_data[19].valid := 1, [93].time.Year := 2022, [93].time.Month := 4, [93].time.Day := 30, [93].time.Hour := 14, [93].time.Minute := 59, [93].time.Second := 59, [93].time.DST_ON := 1, [94].log_data[0].min := 1.0, [94].log_data[0].max := 1.0, [94].log_data[0].total := 3600.0, [94].log_data[0].time := 3600.0, [94].log_data[0].valid := 1, [94].log_data[1].max := 1.0, [94].log_data[1].total := 509.0, [94].log_data[1].time := 3600.0, [94].log_data[1].maxminute := 4, [94].log_data[1].valid := 1, [94].log_data[2].time := 3600.0, [94].log_data[2].valid := 1, [94].log_data[3].time := 3600.0, [94].log_data[3].valid := 1, [94].log_data[4].min := 0.48749998, [94].log_data[4].max := 1.00875, [94].log_data[4].total := 2662.5059, [94].log_data[4].time := 3600.0, [94].log_data[4].minminute := 12, [94].log_data[4].maxminute := 4, [94].log_data[4].valid := 1, [94].log_data[5].max := 7.14, [94].log_data[5].total := 3576.5505, [94].log_data[5].time := 3600.0, [94].log_data[5].maxminute := 5, [94].log_data[5].valid := 1, [94].log_data[6].valid := 1, [94].log_data[7].valid := 1, [94].log_data[8].valid := 1, [94].log_data[9].valid := 1, [94].log_data[10].valid := 1, [94].log_data[11].valid := 1, [94].log_data[12].valid := 1, [94].log_data[13].valid := 1, [94].log_data[14].valid := 1, [94].log_data[15].valid := 1, [94].log_data[16].valid := 1, [94].log_data[17].valid := 1, [94].log_data[18].valid := 1, [94].log_data[19].valid := 1, [94].time.Year := 2022, [94].time.Month := 4, [94].time.Day := 30, [94].time.Hour := 15, [94].time.Minute := 59, [94].time.Second := 59, [94].time.DST_ON := 1, [95].log_data[0].min := 1.0,
        [95].log_data[0].max := 1.0, [95].log_data[0].total := 3599.999, [95].log_data[0].time := 3599.999, [95].log_data[0].valid := 1, [95].log_data[1].time := 3599.999, [95].log_data[1].valid := 1, [95].log_data[2].max := 1.0, [95].log_data[2].total := 491.5, [95].log_data[2].time := 3599.999, [95].log_data[2].maxminute := 30, [95].log_data[2].valid := 1, [95].log_data[3].time := 3599.999, [95].log_data[3].valid := 1, [95].log_data[4].min := 0.48749998, [95].log_data[4].max := 1.00875, [95].log_data[4].total := 2852.676, [95].log_data[4].time := 3599.999, [95].log_data[4].minminute := 38, [95].log_data[4].maxminute := 30, [95].log_data[4].valid := 1, [95].log_data[5].max := 7.23125, [95].log_data[5].total := 3484.0486, [95].log_data[5].time := 3599.999, [95].log_data[5].maxminute := 31, [95].log_data[5].valid := 1, [95].log_data[6].valid := 1, [95].log_data[7].valid := 1, [95].log_data[8].valid := 1, [95].log_data[9].valid := 1, [95].log_data[10].valid := 1, [95].log_data[11].valid := 1, [95].log_data[12].valid := 1, [95].log_data[13].valid := 1, [95].log_data[14].valid := 1, [95].log_data[15].valid := 1, [95].log_data[16].valid := 1, [95].log_data[17].valid := 1, [95].log_data[18].valid := 1, [95].log_data[19].valid := 1, [95].time.Year := 2022, [95].time.Month := 4, [95].time.Day := 30, [95].time.Hour := 16, [95].time.Minute := 59, [95].time.Second := 59, [95].time.DST_ON := 1, [96].log_data[0].min := 1.0, [96].log_data[0].max := 1.0, [96].log_data[0].total := 3600.0, [96].log_data[0].time := 3600.0, [96].log_data[0].valid := 1, [96].log_data[1].time := 3600.0, [96].log_data[1].valid := 1, [96].log_data[2].time := 3600.0, [96].log_data[2].valid := 1, [96].log_data[3].time := 3600.0, [96].log_data[3].valid := 1, [96].log_data[4].min := 0.656875, [96].log_data[4].max := 0.97937495, [96].log_data[4].total := 3100.7124,
        [96].log_data[4].time := 3600.0, [96].log_data[4].maxminute := 56, [96].log_data[4].valid := 1, [96].log_data[5].time := 3600.0, [96].log_data[5].valid := 1, [96].log_data[6].valid := 1, [96].log_data[7].valid := 1, [96].log_data[8].valid := 1, [96].log_data[9].valid := 1, [96].log_data[10].valid := 1, [96].log_data[11].valid := 1, [96].log_data[12].valid := 1, [96].log_data[13].valid := 1, [96].log_data[14].valid := 1, [96].log_data[15].valid := 1, [96].log_data[16].valid := 1, [96].log_data[17].valid := 1, [96].log_data[18].valid := 1, [96].log_data[19].valid := 1, [96].time.Year := 2022, [96].time.Month := 4, [96].time.Day := 30, [96].time.Hour := 17, [96].time.Minute := 59, [96].time.Second := 59, [96].time.DST_ON := 1, [97].log_data[0].min := 1.0, [97].log_data[0].max := 1.0, [97].log_data[0].total := 3600.0, [97].log_data[0].time := 3600.0, [97].log_data[0].valid := 1, [97].log_data[1].max := 1.0, [97].log_data[1].total := 492.0, [97].log_data[1].time := 3600.0, [97].log_data[1].maxminute := 6, [97].log_data[1].valid := 1, [97].log_data[2].time := 3600.0, [97].log_data[2].valid := 1, [97].log_data[3].time := 3600.0, [97].log_data[3].valid := 1, [97].log_data[4].min := 0.48749998, [97].log_data[4].max := 1.00625, [97].log_data[4].total := 2653.0283, [97].log_data[4].time := 3600.0, [97].log_data[4].minminute := 14, [97].log_data[4].maxminute := 6, [97].log_data[4].valid := 1, [97].log_data[5].max := 7.18375, [97].log_data[5].total := 3462.5083, [97].log_data[5].time := 3600.0, [97].log_data[5].maxminute := 7, [97].log_data[5].valid := 1, [97].log_data[6].valid := 1, [97].log_data[7].valid := 1, [97].log_data[8].valid := 1, [97].log_data[9].valid := 1, [97].log_data[10].valid := 1, [97].log_data[11].valid := 1, [97].log_data[12].valid := 1, [97].log_data[13].valid := 1,
        [97].log_data[14].valid := 1, [97].log_data[15].valid := 1, [97].log_data[16].valid := 1, [97].log_data[17].valid := 1, [97].log_data[18].valid := 1, [97].log_data[19].valid := 1, [97].time.Year := 2022, [97].time.Month := 4, [97].time.Day := 30, [97].time.Hour := 18, [97].time.Minute := 59, [97].time.Second := 59, [97].time.DST_ON := 1, [98].log_data[0].min := 1.0, [98].log_data[0].max := 1.0, [98].log_data[0].total := 3599.999, [98].log_data[0].time := 3599.999, [98].log_data[0].valid := 1, [98].log_data[1].time := 3599.999, [98].log_data[1].valid := 1, [98].log_data[2].max := 1.0, [98].log_data[2].total := 512.0, [98].log_data[2].time := 3599.999, [98].log_data[2].maxminute := 18, [98].log_data[2].valid := 1, [98].log_data[3].time := 3599.999, [98].log_data[3].valid := 1, [98].log_data[4].min := 0.48749998, [98].log_data[4].max := 1.00875, [98].log_data[4].total := 2748.1016, [98].log_data[4].time := 3599.999, [98].log_data[4].minminute := 26, [98].log_data[4].maxminute := 18, [98].log_data[4].valid := 1, [98].log_data[5].max := 7.2250004, [98].log_data[5].total := 3631.66, [98].log_data[5].time := 3599.999, [98].log_data[5].maxminute := 18, [98].log_data[5].valid := 1, [98].log_data[6].valid := 1, [98].log_data[7].valid := 1, [98].log_data[8].valid := 1, [98].log_data[9].valid := 1, [98].log_data[10].valid := 1, [98].log_data[11].valid := 1, [98].log_data[12].valid := 1, [98].log_data[13].valid := 1, [98].log_data[14].valid := 1, [98].log_data[15].valid := 1, [98].log_data[16].valid := 1, [98].log_data[17].valid := 1, [98].log_data[18].valid := 1, [98].log_data[19].valid := 1, [98].time.Year := 2022, [98].time.Month := 4, [98].time.Day := 30, [98].time.Hour := 19, [98].time.Minute := 59, [98].time.Second := 59, [98].time.DST_ON := 1,
        [99].log_data[0].min := 1.0, [99].log_data[0].max := 1.0, [99].log_data[0].total := 3600.002, [99].log_data[0].time := 3600.002, [99].log_data[0].valid := 1, [99].log_data[1].max := 1.0, [99].log_data[1].total := 521.0, [99].log_data[1].time := 3600.002, [99].log_data[1].maxminute := 36, [99].log_data[1].valid := 1, [99].log_data[2].time := 3600.002, [99].log_data[2].valid := 1, [99].log_data[3].time := 3600.002, [99].log_data[3].valid := 1, [99].log_data[4].min := 0.48749998, [99].log_data[4].max := 1.00875, [99].log_data[4].total := 2950.3428, [99].log_data[4].time := 3600.002, [99].log_data[4].minminute := 45, [99].log_data[4].maxminute := 36, [99].log_data[4].valid := 1, [99].log_data[5].max := 7.1275, [99].log_data[5].total := 3651.0518, [99].log_data[5].time := 3600.002, [99].log_data[5].maxminute := 37, [99].log_data[5].valid := 1, [99].log_data[6].valid := 1, [99].log_data[7].valid := 1, [99].log_data[8].valid := 1, [99].log_data[9].valid := 1, [99].log_data[10].valid := 1, [99].log_data[11].valid := 1, [99].log_data[12].valid := 1, [99].log_data[13].valid := 1, [99].log_data[14].valid := 1, [99].log_data[15].valid := 1, [99].log_data[16].valid := 1, [99].log_data[17].valid := 1, [99].log_data[18].valid := 1, [99].log_data[19].valid := 1, [99].time.Year := 2022, [99].time.Month := 4, [99].time.Day := 30, [99].time.Hour := 20, [99].time.Minute := 59, [99].time.Second := 59, [99].time.DST_ON := 1, [100].log_data[0].min := 1.0, [100].log_data[0].max := 1.0, [100].log_data[0].total := 3600.0, [100].log_data[0].time := 3600.0, [100].log_data[0].valid := 1, [100].log_data[1].time := 3600.0, [100].log_data[1].valid := 1, [100].log_data[2].max := 1.0, [100].log_data[2].total := 515.0, [100].log_data[2].time := 3600.0, [100].log_data[2].maxminute := 39, [100].log_data[2].valid := 1, [100].log_data[3].time := 3600.0,
        [100].log_data[3].valid := 1, [100].log_data[4].min := 0.48812497, [100].log_data[4].max := 1.00875, [100].log_data[4].total := 2895.3071, [100].log_data[4].time := 3600.0, [100].log_data[4].minminute := 48, [100].log_data[4].maxminute := 39, [100].log_data[4].valid := 1, [100].log_data[5].max := 7.2449994, [100].log_data[5].total := 3655.9912, [100].log_data[5].time := 3600.0, [100].log_data[5].maxminute := 40, [100].log_data[5].valid := 1, [100].log_data[6].valid := 1, [100].log_data[7].valid := 1, [100].log_data[8].valid := 1, [100].log_data[9].valid := 1, [100].log_data[10].valid := 1, [100].log_data[11].valid := 1, [100].log_data[12].valid := 1, [100].log_data[13].valid := 1, [100].log_data[14].valid := 1, [100].log_data[15].valid := 1, [100].log_data[16].valid := 1, [100].log_data[17].valid := 1, [100].log_data[18].valid := 1, [100].log_data[19].valid := 1, [100].time.Year := 2022, [100].time.Month := 4, [100].time.Day := 30, [100].time.Hour := 21, [100].time.Minute := 59, [100].time.Second := 59, [100].time.DST_ON := 1, [101].log_data[0].min := 1.0, [101].log_data[0].max := 1.0, [101].log_data[0].total := 3600.0, [101].log_data[0].time := 3600.0, [101].log_data[0].valid := 1, [101].log_data[1].time := 3600.0, [101].log_data[1].valid := 1, [101].log_data[2].time := 3600.0, [101].log_data[2].valid := 1, [101].log_data[3].time := 3600.0, [101].log_data[3].valid := 1, [101].log_data[4].min := 0.610625, [101].log_data[4].max := 0.995, [101].log_data[4].total := 3035.6504, [101].log_data[4].time := 3600.0, [101].log_data[4].maxminute := 57, [101].log_data[4].valid := 1, [101].log_data[5].max := 0.0012500001, [101].log_data[5].total := 1.0393883, [101].log_data[5].time := 3600.0, [101].log_data[5].valid := 1, [101].log_data[6].valid := 1, [101].log_data[7].valid := 1, [101].log_data[8].valid := 1, [101].log_data[9].valid := 1, [101].log_data[10].valid := 1,
        [101].log_data[11].valid := 1, [101].log_data[12].valid := 1, [101].log_data[13].valid := 1, [101].log_data[14].valid := 1, [101].log_data[15].valid := 1, [101].log_data[16].valid := 1, [101].log_data[17].valid := 1, [101].log_data[18].valid := 1, [101].log_data[19].valid := 1, [101].time.Year := 2022, [101].time.Month := 4, [101].time.Day := 30, [101].time.Hour := 22, [101].time.Minute := 59, [101].time.Second := 59, [101].time.DST_ON := 1, [102].log_data[0].min := 1.0, [102].log_data[0].max := 1.0, [102].log_data[0].total := 3600.0, [102].log_data[0].time := 3600.0, [102].log_data[0].valid := 1, [102].log_data[1].max := 1.0, [102].log_data[1].total := 498.0, [102].log_data[1].time := 3600.0, [102].log_data[1].maxminute := 1, [102].log_data[1].valid := 1, [102].log_data[2].time := 3600.0, [102].log_data[2].valid := 1, [102].log_data[3].time := 3600.0, [102].log_data[3].valid := 1, [102].log_data[4].min := 0.48812497, [102].log_data[4].max := 1.005625, [102].log_data[4].total := 2670.1338, [102].log_data[4].time := 3600.0, [102].log_data[4].minminute := 10, [102].log_data[4].maxminute := 1, [102].log_data[4].valid := 1, [102].log_data[5].max := 7.133749, [102].log_data[5].total := 3495.4927, [102].log_data[5].time := 3600.0, [102].log_data[5].maxminute := 2, [102].log_data[5].valid := 1, [102].log_data[6].valid := 1, [102].log_data[7].valid := 1, [102].log_data[8].valid := 1, [102].log_data[9].valid := 1, [102].log_data[10].valid := 1, [102].log_data[11].valid := 1, [102].log_data[12].valid := 1, [102].log_data[13].valid := 1, [102].log_data[14].valid := 1, [102].log_data[15].valid := 1, [102].log_data[16].valid := 1, [102].log_data[17].valid := 1, [102].log_data[18].valid := 1, [102].log_data[19].valid := 1, [102].time.Year := 2022, [102].time.Month := 4, [102].time.Day := 30, [102].time.Hour := 23,
        [102].time.Minute := 59, [102].time.Second := 59, [102].time.DST_ON := 1, [103].log_data[0].min := 1.0, [103].log_data[0].max := 1.0, [103].log_data[0].total := 3600.0, [103].log_data[0].time := 3600.0, [103].log_data[0].valid := 1, [103].log_data[1].time := 3600.0, [103].log_data[1].valid := 1, [103].log_data[2].max := 1.0, [103].log_data[2].total := 486.499, [103].log_data[2].time := 3600.0, [103].log_data[2].maxminute := 28, [103].log_data[2].valid := 1, [103].log_data[3].time := 3600.0, [103].log_data[3].valid := 1, [103].log_data[4].min := 0.48812497, [103].log_data[4].max := 1.00125, [103].log_data[4].total := 2807.5156, [103].log_data[4].time := 3600.0, [103].log_data[4].minminute := 36, [103].log_data[4].maxminute := 28, [103].log_data[4].valid := 1, [103].log_data[5].max := 7.2912507, [103].log_data[5].total := 3484.4834, [103].log_data[5].time := 3600.0, [103].log_data[5].maxminute := 29, [103].log_data[5].valid := 1, [103].log_data[6].valid := 1, [103].log_data[7].valid := 1, [103].log_data[8].valid := 1, [103].log_data[9].valid := 1, [103].log_data[10].valid := 1, [103].log_data[11].valid := 1, [103].log_data[12].valid := 1, [103].log_data[13].valid := 1, [103].log_data[14].valid := 1, [103].log_data[15].valid := 1, [103].log_data[16].valid := 1, [103].log_data[17].valid := 1, [103].log_data[18].valid := 1, [103].log_data[19].valid := 1, [103].time.Year := 2022, [103].time.Month := 5, [103].time.Day := 1, [103].time.Minute := 59, [103].time.Second := 59, [103].time.DST_ON := 1, [104].log_data[0].min := 1.0, [104].log_data[0].max := 1.0, [104].log_data[0].total := 3600.0, [104].log_data[0].time := 3600.0, [104].log_data[0].valid := 1, [104].log_data[1].time := 3600.0, [104].log_data[1].valid := 1, [104].log_data[2].time := 3600.0, [104].log_data[2].valid := 1, [104].log_data[3].time := 3600.0, [104].log_data[3].valid := 1,
        [104].log_data[4].min := 0.62624997, [104].log_data[4].max := 0.91875005, [104].log_data[4].total := 2830.3225, [104].log_data[4].time := 3600.0, [104].log_data[4].maxminute := 59, [104].log_data[4].valid := 1, [104].log_data[5].max := 0.0012500001, [104].log_data[5].total := 1.4030772, [104].log_data[5].time := 3600.0, [104].log_data[5].valid := 1, [104].log_data[6].valid := 1, [104].log_data[7].valid := 1, [104].log_data[8].valid := 1, [104].log_data[9].valid := 1, [104].log_data[10].valid := 1, [104].log_data[11].valid := 1, [104].log_data[12].valid := 1, [104].log_data[13].valid := 1, [104].log_data[14].valid := 1, [104].log_data[15].valid := 1, [104].log_data[16].valid := 1, [104].log_data[17].valid := 1, [104].log_data[18].valid := 1, [104].log_data[19].valid := 1, [104].time.Year := 2022, [104].time.Month := 5, [104].time.Day := 1, [104].time.Hour := 1, [104].time.Minute := 59, [104].time.Second := 59, [104].time.DST_ON := 1, [105].log_data[0].min := 1.0, [105].log_data[0].max := 1.0, [105].log_data[0].total := 3600.0, [105].log_data[0].time := 3600.0, [105].log_data[0].valid := 1, [105].log_data[1].max := 1.0, [105].log_data[1].total := 478.0, [105].log_data[1].time := 3600.0, [105].log_data[1].maxminute := 51, [105].log_data[1].valid := 1, [105].log_data[2].time := 3600.0, [105].log_data[2].valid := 1, [105].log_data[3].time := 3600.0, [105].log_data[3].valid := 1, [105].log_data[4].min := 0.48812497, [105].log_data[4].max := 1.0068749, [105].log_data[4].total := 3375.1597, [105].log_data[4].time := 3600.0, [105].log_data[4].minminute := 59, [105].log_data[4].maxminute := 51, [105].log_data[4].valid := 1, [105].log_data[5].max := 7.1512504, [105].log_data[5].total := 3358.7073, [105].log_data[5].time := 3600.0, [105].log_data[5].maxminute := 52, [105].log_data[5].valid := 1, [105].log_data[6].valid := 1, [105].log_data[7].valid := 1, [105].log_data[8].valid := 1,
        [105].log_data[9].valid := 1, [105].log_data[10].valid := 1, [105].log_data[11].valid := 1, [105].log_data[12].valid := 1, [105].log_data[13].valid := 1, [105].log_data[14].valid := 1, [105].log_data[15].valid := 1, [105].log_data[16].valid := 1, [105].log_data[17].valid := 1, [105].log_data[18].valid := 1, [105].log_data[19].valid := 1, [105].time.Year := 2022, [105].time.Month := 5, [105].time.Day := 1, [105].time.Hour := 2, [105].time.Minute := 59, [105].time.Second := 59, [105].time.DST_ON := 1, [106].log_data[0].min := 1.0, [106].log_data[0].max := 1.0, [106].log_data[0].total := 3599.999, [106].log_data[0].time := 3599.999, [106].log_data[0].valid := 1, [106].log_data[1].time := 3599.999, [106].log_data[1].valid := 1, [106].log_data[2].time := 3599.999, [106].log_data[2].valid := 1, [106].log_data[3].time := 3599.999, [106].log_data[3].valid := 1, [106].log_data[4].min := 0.48812497, [106].log_data[4].max := 0.68875, [106].log_data[4].total := 2135.9, [106].log_data[4].time := 3599.999, [106].log_data[4].maxminute := 57, [106].log_data[4].valid := 1, [106].log_data[5].max := 0.0025000002, [106].log_data[5].total := 2.6781197, [106].log_data[5].time := 3599.999, [106].log_data[5].maxminute := 28, [106].log_data[5].valid := 1, [106].log_data[6].valid := 1, [106].log_data[7].valid := 1, [106].log_data[8].valid := 1, [106].log_data[9].valid := 1, [106].log_data[10].valid := 1, [106].log_data[11].valid := 1, [106].log_data[12].valid := 1, [106].log_data[13].valid := 1, [106].log_data[14].valid := 1, [106].log_data[15].valid := 1, [106].log_data[16].valid := 1, [106].log_data[17].valid := 1, [106].log_data[18].valid := 1, [106].log_data[19].valid := 1, [106].time.Year := 2022, [106].time.Month := 5, [106].time.Day := 1, [106].time.Hour := 3, [106].time.Minute := 59, [106].time.Second := 59,
        [106].time.DST_ON := 1, [107].log_data[0].min := 1.0, [107].log_data[0].max := 1.0, [107].log_data[0].total := 3599.999, [107].log_data[0].time := 3599.999, [107].log_data[0].valid := 1, [107].log_data[1].time := 3599.999, [107].log_data[1].valid := 1, [107].log_data[2].time := 3599.999, [107].log_data[2].valid := 1, [107].log_data[3].time := 3599.999, [107].log_data[3].valid := 1, [107].log_data[4].min := 0.68812495, [107].log_data[4].max := 0.8268749, [107].log_data[4].total := 2733.8613, [107].log_data[4].time := 3599.999, [107].log_data[4].maxminute := 55, [107].log_data[4].valid := 1, [107].log_data[5].max := 0.0012500001, [107].log_data[5].total := 2.7178178, [107].log_data[5].time := 3599.999, [107].log_data[5].valid := 1, [107].log_data[6].valid := 1, [107].log_data[7].valid := 1, [107].log_data[8].valid := 1, [107].log_data[9].valid := 1, [107].log_data[10].valid := 1, [107].log_data[11].valid := 1, [107].log_data[12].valid := 1, [107].log_data[13].valid := 1, [107].log_data[14].valid := 1, [107].log_data[15].valid := 1, [107].log_data[16].valid := 1, [107].log_data[17].valid := 1, [107].log_data[18].valid := 1, [107].log_data[19].valid := 1, [107].time.Year := 2022, [107].time.Month := 5, [107].time.Day := 1, [107].time.Hour := 4, [107].time.Minute := 59, [107].time.Second := 59, [107].time.DST_ON := 1, [108].log_data[0].min := 1.0, [108].log_data[0].max := 1.0, [108].log_data[0].total := 3599.999, [108].log_data[0].time := 3599.999, [108].log_data[0].valid := 1, [108].log_data[1].time := 3599.999, [108].log_data[1].valid := 1, [108].log_data[2].time := 3599.999, [108].log_data[2].valid := 1, [108].log_data[3].time := 3599.999, [108].log_data[3].valid := 1, [108].log_data[4].min := 0.82625, [108].log_data[4].max := 0.91875005, [108].log_data[4].total := 3165.775, [108].log_data[4].time := 3599.999, [108].log_data[4].maxminute := 54, [108].log_data[4].valid := 1,
        [108].log_data[5].max := 0.0025000002, [108].log_data[5].total := 3.2923117, [108].log_data[5].time := 3599.999, [108].log_data[5].maxminute := 42, [108].log_data[5].valid := 1, [108].log_data[6].valid := 1, [108].log_data[7].valid := 1, [108].log_data[8].valid := 1, [108].log_data[9].valid := 1, [108].log_data[10].valid := 1, [108].log_data[11].valid := 1, [108].log_data[12].valid := 1, [108].log_data[13].valid := 1, [108].log_data[14].valid := 1, [108].log_data[15].valid := 1, [108].log_data[16].valid := 1, [108].log_data[17].valid := 1, [108].log_data[18].valid := 1, [108].log_data[19].valid := 1, [108].time.Year := 2022, [108].time.Month := 5, [108].time.Day := 1, [108].time.Hour := 5, [108].time.Minute := 59, [108].time.Second := 59, [108].time.DST_ON := 1, [109].log_data[0].min := 1.0, [109].log_data[0].max := 1.0, [109].log_data[0].total := 3600.0, [109].log_data[0].time := 3600.0, [109].log_data[0].valid := 1, [109].log_data[1].time := 3600.0, [109].log_data[1].valid := 1, [109].log_data[2].time := 3600.0, [109].log_data[2].valid := 1, [109].log_data[3].time := 3600.0, [109].log_data[3].valid := 1, [109].log_data[4].min := 0.91875005, [109].log_data[4].max := 0.94875, [109].log_data[4].total := 3372.2683, [109].log_data[4].time := 3600.0, [109].log_data[4].maxminute := 36, [109].log_data[4].valid := 1, [109].log_data[5].max := 0.0025000002, [109].log_data[5].total := 3.1313436, [109].log_data[5].time := 3600.0, [109].log_data[5].valid := 1, [109].log_data[6].valid := 1, [109].log_data[7].valid := 1, [109].log_data[8].valid := 1, [109].log_data[9].valid := 1, [109].log_data[10].valid := 1, [109].log_data[11].valid := 1, [109].log_data[12].valid := 1, [109].log_data[13].valid := 1, [109].log_data[14].valid := 1, [109].log_data[15].valid := 1, [109].log_data[16].valid := 1, [109].log_data[17].valid := 1, [109].log_data[18].valid := 1,
        [109].log_data[19].valid := 1, [109].time.Year := 2022, [109].time.Month := 5, [109].time.Day := 1, [109].time.Hour := 6, [109].time.Minute := 59, [109].time.Second := 59, [109].time.DST_ON := 1, [110].log_data[0].min := 1.0, [110].log_data[0].max := 1.0, [110].log_data[0].total := 3600.0, [110].log_data[0].time := 3600.0, [110].log_data[0].valid := 1, [110].log_data[1].time := 3600.0, [110].log_data[1].valid := 1, [110].log_data[2].time := 3600.0, [110].log_data[2].valid := 1, [110].log_data[3].time := 3600.0, [110].log_data[3].valid := 1, [110].log_data[4].min := 0.94875, [110].log_data[4].max := 0.98, [110].log_data[4].total := 3484.1028, [110].log_data[4].time := 3600.0, [110].log_data[4].maxminute := 41, [110].log_data[4].valid := 1, [110].log_data[5].max := 0.0012500001, [110].log_data[5].total := 2.4230673, [110].log_data[5].time := 3600.0, [110].log_data[5].valid := 1, [110].log_data[6].valid := 1, [110].log_data[7].valid := 1, [110].log_data[8].valid := 1, [110].log_data[9].valid := 1, [110].log_data[10].valid := 1, [110].log_data[11].valid := 1, [110].log_data[12].valid := 1, [110].log_data[13].valid := 1, [110].log_data[14].valid := 1, [110].log_data[15].valid := 1, [110].log_data[16].valid := 1, [110].log_data[17].valid := 1, [110].log_data[18].valid := 1, [110].log_data[19].valid := 1, [110].time.Year := 2022, [110].time.Month := 5, [110].time.Day := 1, [110].time.Hour := 7, [110].time.Minute := 59, [110].time.Second := 59, [110].time.DST_ON := 1, [111].log_data[0].min := 1.0, [111].log_data[0].max := 1.0, [111].log_data[0].total := 3600.0, [111].log_data[0].time := 3600.0, [111].log_data[0].valid := 1, [111].log_data[1].time := 3600.0, [111].log_data[1].valid := 1, [111].log_data[2].max := 1.0, [111].log_data[2].total := 481.0, [111].log_data[2].time := 3600.0,
        [111].log_data[2].maxminute := 21, [111].log_data[2].valid := 1, [111].log_data[3].time := 3600.0, [111].log_data[3].valid := 1, [111].log_data[4].min := 0.48812497, [111].log_data[4].max := 1.0024999, [111].log_data[4].total := 2741.4768, [111].log_data[4].time := 3600.0, [111].log_data[4].minminute := 30, [111].log_data[4].maxminute := 21, [111].log_data[4].valid := 1, [111].log_data[5].max := 7.25375, [111].log_data[5].total := 3424.0884, [111].log_data[5].time := 3600.0, [111].log_data[5].maxminute := 23, [111].log_data[5].valid := 1, [111].log_data[6].valid := 1, [111].log_data[7].valid := 1, [111].log_data[8].valid := 1, [111].log_data[9].valid := 1, [111].log_data[10].valid := 1, [111].log_data[11].valid := 1, [111].log_data[12].valid := 1, [111].log_data[13].valid := 1, [111].log_data[14].valid := 1, [111].log_data[15].valid := 1, [111].log_data[16].valid := 1, [111].log_data[17].valid := 1, [111].log_data[18].valid := 1, [111].log_data[19].valid := 1, [111].time.Year := 2022, [111].time.Month := 5, [111].time.Day := 1, [111].time.Hour := 8, [111].time.Minute := 59, [111].time.Second := 59, [111].time.DST_ON := 1, [112].log_data[0].min := 1.0, [112].log_data[0].max := 1.0, [112].log_data[0].total := 3600.0, [112].log_data[0].time := 3600.0, [112].log_data[0].valid := 1, [112].log_data[1].max := 1.0, [112].log_data[1].total := 57.75, [112].log_data[1].time := 3600.0, [112].log_data[1].maxminute := 59, [112].log_data[1].valid := 1, [112].log_data[2].time := 3600.0, [112].log_data[2].valid := 1, [112].log_data[3].time := 3600.0, [112].log_data[3].valid := 1, [112].log_data[4].min := 0.686875, [112].log_data[4].max := 1.00875, [112].log_data[4].total := 3062.8977, [112].log_data[4].time := 3600.0, [112].log_data[4].maxminute := 59, [112].log_data[4].valid := 1, [112].log_data[5].max := 7.1512504, [112].log_data[5].total := 353.88962, [112].log_data[5].time := 3600.0,
        [112].log_data[5].maxminute := 59, [112].log_data[5].valid := 1, [112].log_data[6].valid := 1, [112].log_data[7].valid := 1, [112].log_data[8].valid := 1, [112].log_data[9].valid := 1, [112].log_data[10].valid := 1, [112].log_data[11].valid := 1, [112].log_data[12].valid := 1, [112].log_data[13].valid := 1, [112].log_data[14].valid := 1, [112].log_data[15].valid := 1, [112].log_data[16].valid := 1, [112].log_data[17].valid := 1, [112].log_data[18].valid := 1, [112].log_data[19].valid := 1, [112].time.Year := 2022, [112].time.Month := 5, [112].time.Day := 1, [112].time.Hour := 9, [112].time.Minute := 59, [112].time.Second := 59, [112].time.DST_ON := 1, [113].log_data[0].min := 1.0, [113].log_data[0].max := 1.0, [113].log_data[0].total := 3600.0, [113].log_data[0].time := 3600.0, [113].log_data[0].valid := 1, [113].log_data[1].max := 1.0, [113].log_data[1].total := 465.75, [113].log_data[1].time := 3600.0, [113].log_data[1].minminute := 7, [113].log_data[1].valid := 1, [113].log_data[2].time := 3600.0, [113].log_data[2].valid := 1, [113].log_data[3].time := 3600.0, [113].log_data[3].valid := 1, [113].log_data[4].min := 0.48812497, [113].log_data[4].max := 0.995, [113].log_data[4].total := 2780.916, [113].log_data[4].time := 3600.0, [113].log_data[4].minminute := 7, [113].log_data[4].maxminute := 59, [113].log_data[4].valid := 1, [113].log_data[5].max := 7.1475, [113].log_data[5].total := 3328.9827, [113].log_data[5].time := 3600.0, [113].log_data[5].minminute := 8, [113].log_data[5].valid := 1, [113].log_data[6].valid := 1, [113].log_data[7].valid := 1, [113].log_data[8].valid := 1, [113].log_data[9].valid := 1, [113].log_data[10].valid := 1, [113].log_data[11].valid := 1, [113].log_data[12].valid := 1, [113].log_data[13].valid := 1, [113].log_data[14].valid := 1, [113].log_data[15].valid := 1, [113].log_data[16].valid := 1,
        [113].log_data[17].valid := 1, [113].log_data[18].valid := 1, [113].log_data[19].valid := 1, [113].time.Year := 2022, [113].time.Month := 5, [113].time.Day := 1, [113].time.Hour := 10, [113].time.Minute := 59, [113].time.Second := 59, [113].time.DST_ON := 1, [114].log_data[0].min := 1.0, [114].log_data[0].max := 1.0, [114].log_data[0].total := 3600.0, [114].log_data[0].time := 3600.0, [114].log_data[0].valid := 1, [114].log_data[1].time := 3600.0, [114].log_data[1].valid := 1, [114].log_data[2].max := 1.0, [114].log_data[2].total := 515.0, [114].log_data[2].time := 3600.0, [114].log_data[2].maxminute := 1, [114].log_data[2].valid := 1, [114].log_data[3].time := 3600.0, [114].log_data[3].valid := 1, [114].log_data[4].min := 0.48812497, [114].log_data[4].max := 1.00875, [114].log_data[4].total := 2797.7185, [114].log_data[4].time := 3600.0, [114].log_data[4].minminute := 10, [114].log_data[4].maxminute := 1, [114].log_data[4].valid := 1, [114].log_data[5].max := 7.2425003, [114].log_data[5].total := 3665.3699, [114].log_data[5].time := 3600.0, [114].log_data[5].maxminute := 2, [114].log_data[5].valid := 1, [114].log_data[6].valid := 1, [114].log_data[7].valid := 1, [114].log_data[8].valid := 1, [114].log_data[9].valid := 1, [114].log_data[10].valid := 1, [114].log_data[11].valid := 1, [114].log_data[12].valid := 1, [114].log_data[13].valid := 1, [114].log_data[14].valid := 1, [114].log_data[15].valid := 1, [114].log_data[16].valid := 1, [114].log_data[17].valid := 1, [114].log_data[18].valid := 1, [114].log_data[19].valid := 1, [114].time.Year := 2022, [114].time.Month := 5, [114].time.Day := 1, [114].time.Hour := 11, [114].time.Minute := 59, [114].time.Second := 59, [114].time.DST_ON := 1, [115].log_data[0].min := 1.0, [115].log_data[0].max := 1.0, [115].log_data[0].total := 3600.0,
        [115].log_data[0].time := 3600.0, [115].log_data[0].valid := 1, [115].log_data[1].max := 1.0, [115].log_data[1].total := 524.0, [115].log_data[1].time := 3600.0, [115].log_data[1].maxminute := 5, [115].log_data[1].valid := 1, [115].log_data[2].time := 3600.0, [115].log_data[2].valid := 1, [115].log_data[3].time := 3600.0, [115].log_data[3].valid := 1, [115].log_data[4].min := 0.48749998, [115].log_data[4].max := 1.00875, [115].log_data[4].total := 2871.14, [115].log_data[4].time := 3600.0, [115].log_data[4].minminute := 14, [115].log_data[4].maxminute := 5, [115].log_data[4].valid := 1, [115].log_data[5].max := 7.1512504, [115].log_data[5].total := 3677.105, [115].log_data[5].time := 3600.0, [115].log_data[5].maxminute := 6, [115].log_data[5].valid := 1, [115].log_data[6].valid := 1, [115].log_data[7].valid := 1, [115].log_data[8].valid := 1, [115].log_data[9].valid := 1, [115].log_data[10].valid := 1, [115].log_data[11].valid := 1, [115].log_data[12].valid := 1, [115].log_data[13].valid := 1, [115].log_data[14].valid := 1, [115].log_data[15].valid := 1, [115].log_data[16].valid := 1, [115].log_data[17].valid := 1, [115].log_data[18].valid := 1, [115].log_data[19].valid := 1, [115].time.Year := 2022, [115].time.Month := 5, [115].time.Day := 1, [115].time.Hour := 12, [115].time.Minute := 59, [115].time.Second := 59, [115].time.DST_ON := 1, [116].log_data[0].min := 1.0, [116].log_data[0].max := 1.0, [116].log_data[0].total := 3600.0, [116].log_data[0].time := 3600.0, [116].log_data[0].valid := 1, [116].log_data[1].time := 3600.0, [116].log_data[1].valid := 1, [116].log_data[2].max := 1.0, [116].log_data[2].total := 510.0, [116].log_data[2].time := 3600.0, [116].log_data[2].maxminute := 9, [116].log_data[2].valid := 1, [116].log_data[3].time := 3600.0, [116].log_data[3].valid := 1, [116].log_data[4].min := 0.48749998, [116].log_data[4].max := 1.0068749,
        [116].log_data[4].total := 2743.2285, [116].log_data[4].time := 3600.0, [116].log_data[4].minminute := 18, [116].log_data[4].maxminute := 9, [116].log_data[4].valid := 1, [116].log_data[5].max := 7.23125, [116].log_data[5].total := 3619.7273, [116].log_data[5].time := 3600.0, [116].log_data[5].maxminute := 12, [116].log_data[5].valid := 1, [116].log_data[6].valid := 1, [116].log_data[7].valid := 1, [116].log_data[8].valid := 1, [116].log_data[9].valid := 1, [116].log_data[10].valid := 1, [116].log_data[11].valid := 1, [116].log_data[12].valid := 1, [116].log_data[13].valid := 1, [116].log_data[14].valid := 1, [116].log_data[15].valid := 1, [116].log_data[16].valid := 1, [116].log_data[17].valid := 1, [116].log_data[18].valid := 1, [116].log_data[19].valid := 1, [116].time.Year := 2022, [116].time.Month := 5, [116].time.Day := 1, [116].time.Hour := 13, [116].time.Minute := 59, [116].time.Second := 59, [116].time.DST_ON := 1, [117].log_data[0].min := 1.0, [117].log_data[0].max := 1.0, [117].log_data[0].total := 3600.0, [117].log_data[0].time := 3600.0, [117].log_data[0].valid := 1, [117].log_data[1].max := 1.0, [117].log_data[1].total := 495.0, [117].log_data[1].time := 3600.0, [117].log_data[1].maxminute := 35, [117].log_data[1].valid := 1, [117].log_data[2].time := 3600.0, [117].log_data[2].valid := 1, [117].log_data[3].time := 3600.0, [117].log_data[3].valid := 1, [117].log_data[4].min := 0.48749998, [117].log_data[4].max := 1.0074999, [117].log_data[4].total := 2955.6804, [117].log_data[4].time := 3600.0, [117].log_data[4].minminute := 44, [117].log_data[4].maxminute := 36, [117].log_data[4].valid := 1, [117].log_data[5].max := 7.1675005, [117].log_data[5].total := 3474.0054, [117].log_data[5].time := 3600.0, [117].log_data[5].maxminute := 36, [117].log_data[5].valid := 1, [117].log_data[6].valid := 1, [117].log_data[7].valid := 1, [117].log_data[8].valid := 1,
        [117].log_data[9].valid := 1, [117].log_data[10].valid := 1, [117].log_data[11].valid := 1, [117].log_data[12].valid := 1, [117].log_data[13].valid := 1, [117].log_data[14].valid := 1, [117].log_data[15].valid := 1, [117].log_data[16].valid := 1, [117].log_data[17].valid := 1, [117].log_data[18].valid := 1, [117].log_data[19].valid := 1, [117].time.Year := 2022, [117].time.Month := 5, [117].time.Day := 1, [117].time.Hour := 14, [117].time.Minute := 59, [117].time.Second := 59, [117].time.DST_ON := 1, [118].log_data[0].min := 1.0, [118].log_data[0].max := 1.0, [118].log_data[0].total := 3600.0, [118].log_data[0].time := 3600.0, [118].log_data[0].valid := 1, [118].log_data[1].time := 3600.0, [118].log_data[1].valid := 1, [118].log_data[2].time := 3600.0, [118].log_data[2].valid := 1, [118].log_data[3].time := 3600.0, [118].log_data[3].valid := 1, [118].log_data[4].min := 0.595, [118].log_data[4].max := 0.918125, [118].log_data[4].total := 2823.9055, [118].log_data[4].time := 3600.0, [118].log_data[4].maxminute := 55, [118].log_data[4].valid := 1, [118].log_data[5].time := 3600.0, [118].log_data[5].valid := 1, [118].log_data[6].valid := 1, [118].log_data[7].valid := 1, [118].log_data[8].valid := 1, [118].log_data[9].valid := 1, [118].log_data[10].valid := 1, [118].log_data[11].valid := 1, [118].log_data[12].valid := 1, [118].log_data[13].valid := 1, [118].log_data[14].valid := 1, [118].log_data[15].valid := 1, [118].log_data[16].valid := 1, [118].log_data[17].valid := 1, [118].log_data[18].valid := 1, [118].log_data[19].valid := 1, [118].time.Year := 2022, [118].time.Month := 5, [118].time.Day := 1, [118].time.Hour := 15, [118].time.Minute := 59, [118].time.Second := 59, [118].time.DST_ON := 1, [119].log_data[0].min := 1.0, [119].log_data[0].max := 1.0,
        [119].log_data[0].total := 3600.0, [119].log_data[0].time := 3600.0, [119].log_data[0].valid := 1, [119].log_data[1].time := 3600.0, [119].log_data[1].valid := 1, [119].log_data[2].max := 1.0, [119].log_data[2].total := 489.0, [119].log_data[2].time := 3600.0, [119].log_data[2].maxminute := 33, [119].log_data[2].valid := 1, [119].log_data[3].time := 3600.0, [119].log_data[3].valid := 1, [119].log_data[4].min := 0.48687503, [119].log_data[4].max := 1.0024999, [119].log_data[4].total := 2924.6716, [119].log_data[4].time := 3600.0, [119].log_data[4].minminute := 42, [119].log_data[4].maxminute := 33, [119].log_data[4].valid := 1, [119].log_data[5].max := 7.2237496, [119].log_data[5].total := 3464.3586, [119].log_data[5].time := 3600.0, [119].log_data[5].maxminute := 34, [119].log_data[5].valid := 1, [119].log_data[6].valid := 1, [119].log_data[7].valid := 1, [119].log_data[8].valid := 1, [119].log_data[9].valid := 1, [119].log_data[10].valid := 1, [119].log_data[11].valid := 1, [119].log_data[12].valid := 1, [119].log_data[13].valid := 1, [119].log_data[14].valid := 1, [119].log_data[15].valid := 1, [119].log_data[16].valid := 1, [119].log_data[17].valid := 1, [119].log_data[18].valid := 1, [119].log_data[19].valid := 1, [119].time.Year := 2022, [119].time.Month := 5, [119].time.Day := 1, [119].time.Hour := 16, [119].time.Minute := 59, [119].time.Second := 59, [119].time.DST_ON := 1, [120].log_data[0].min := 1.0, [120].log_data[0].max := 1.0, [120].log_data[0].total := 3599.999, [120].log_data[0].time := 3599.999, [120].log_data[0].valid := 1, [120].log_data[1].time := 3599.999, [120].log_data[1].valid := 1, [120].log_data[2].time := 3599.999, [120].log_data[2].valid := 1, [120].log_data[3].time := 3599.999, [120].log_data[3].valid := 1, [120].log_data[4].min := 0.61, [120].log_data[4].max := 0.9637501, [120].log_data[4].total := 2941.7788, [120].log_data[4].time := 3599.999,
        [120].log_data[4].maxminute := 59, [120].log_data[4].valid := 1, [120].log_data[5].time := 3599.999, [120].log_data[5].valid := 1, [120].log_data[6].valid := 1, [120].log_data[7].valid := 1, [120].log_data[8].valid := 1, [120].log_data[9].valid := 1, [120].log_data[10].valid := 1, [120].log_data[11].valid := 1, [120].log_data[12].valid := 1, [120].log_data[13].valid := 1, [120].log_data[14].valid := 1, [120].log_data[15].valid := 1, [120].log_data[16].valid := 1, [120].log_data[17].valid := 1, [120].log_data[18].valid := 1, [120].log_data[19].valid := 1, [120].time.Year := 2022, [120].time.Month := 5, [120].time.Day := 1, [120].time.Hour := 17, [120].time.Minute := 59, [120].time.Second := 59, [120].time.DST_ON := 1, [121].log_data[0].min := 1.0, [121].log_data[0].max := 1.0, [121].log_data[0].total := 3600.0, [121].log_data[0].time := 3600.0, [121].log_data[0].valid := 1, [121].log_data[1].max := 1.0, [121].log_data[1].total := 509.0, [121].log_data[1].time := 3600.0, [121].log_data[1].maxminute := 10, [121].log_data[1].valid := 1, [121].log_data[2].time := 3600.0, [121].log_data[2].valid := 1, [121].log_data[3].time := 3600.0, [121].log_data[3].valid := 1, [121].log_data[4].min := 0.48687503, [121].log_data[4].max := 1.0081251, [121].log_data[4].total := 2681.2053, [121].log_data[4].time := 3600.0, [121].log_data[4].minminute := 19, [121].log_data[4].maxminute := 10, [121].log_data[4].valid := 1, [121].log_data[5].max := 7.1300006, [121].log_data[5].total := 3569.1235, [121].log_data[5].time := 3600.0, [121].log_data[5].maxminute := 11, [121].log_data[5].valid := 1, [121].log_data[6].valid := 1, [121].log_data[7].valid := 1, [121].log_data[8].valid := 1, [121].log_data[9].valid := 1, [121].log_data[10].valid := 1, [121].log_data[11].valid := 1, [121].log_data[12].valid := 1, [121].log_data[13].valid := 1, [121].log_data[14].valid := 1,
        [121].log_data[15].valid := 1, [121].log_data[16].valid := 1, [121].log_data[17].valid := 1, [121].log_data[18].valid := 1, [121].log_data[19].valid := 1, [121].time.Year := 2022, [121].time.Month := 5, [121].time.Day := 1, [121].time.Hour := 18, [121].time.Minute := 59, [121].time.Second := 59, [121].time.DST_ON := 1, [122].log_data[0].min := 1.0, [122].log_data[0].max := 1.0, [122].log_data[0].total := 3600.0, [122].log_data[0].time := 3600.0, [122].log_data[0].valid := 1, [122].log_data[1].time := 3600.0, [122].log_data[1].valid := 1, [122].log_data[2].max := 1.0, [122].log_data[2].total := 512.5, [122].log_data[2].time := 3600.0, [122].log_data[2].maxminute := 28, [122].log_data[2].valid := 1, [122].log_data[3].time := 3600.0, [122].log_data[3].valid := 1, [122].log_data[4].min := 0.48749998, [122].log_data[4].max := 1.0081251, [122].log_data[4].total := 2837.2197, [122].log_data[4].time := 3600.0, [122].log_data[4].minminute := 37, [122].log_data[4].maxminute := 28, [122].log_data[4].valid := 1, [122].log_data[5].max := 7.215, [122].log_data[5].total := 3633.7036, [122].log_data[5].time := 3600.0, [122].log_data[5].maxminute := 29, [122].log_data[5].valid := 1, [122].log_data[6].valid := 1, [122].log_data[7].valid := 1, [122].log_data[8].valid := 1, [122].log_data[9].valid := 1, [122].log_data[10].valid := 1, [122].log_data[11].valid := 1, [122].log_data[12].valid := 1, [122].log_data[13].valid := 1, [122].log_data[14].valid := 1, [122].log_data[15].valid := 1, [122].log_data[16].valid := 1, [122].log_data[17].valid := 1, [122].log_data[18].valid := 1, [122].log_data[19].valid := 1, [122].time.Year := 2022, [122].time.Month := 5, [122].time.Day := 1, [122].time.Hour := 19, [122].time.Minute := 59, [122].time.Second := 59, [122].time.DST_ON := 1, [123].log_data[0].min := 1.0,
        [123].log_data[0].max := 1.0, [123].log_data[0].total := 3600.0, [123].log_data[0].time := 3600.0, [123].log_data[0].valid := 1, [123].log_data[1].max := 1.0, [123].log_data[1].total := 506.0, [123].log_data[1].time := 3600.0, [123].log_data[1].maxminute := 40, [123].log_data[1].valid := 1, [123].log_data[2].time := 3600.0, [123].log_data[2].valid := 1, [123].log_data[3].time := 3600.0, [123].log_data[3].valid := 1, [123].log_data[4].min := 0.48749998, [123].log_data[4].max := 1.00875, [123].log_data[4].total := 2947.3635, [123].log_data[4].time := 3600.0, [123].log_data[4].minminute := 49, [123].log_data[4].maxminute := 40, [123].log_data[4].valid := 1, [123].log_data[5].max := 7.13875, [123].log_data[5].total := 3554.1104, [123].log_data[5].time := 3600.0, [123].log_data[5].maxminute := 41, [123].log_data[5].valid := 1, [123].log_data[6].valid := 1, [123].log_data[7].valid := 1, [123].log_data[8].valid := 1, [123].log_data[9].valid := 1, [123].log_data[10].valid := 1, [123].log_data[11].valid := 1, [123].log_data[12].valid := 1, [123].log_data[13].valid := 1, [123].log_data[14].valid := 1, [123].log_data[15].valid := 1, [123].log_data[16].valid := 1, [123].log_data[17].valid := 1, [123].log_data[18].valid := 1, [123].log_data[19].valid := 1, [123].time.Year := 2022, [123].time.Month := 5, [123].time.Day := 1, [123].time.Hour := 20, [123].time.Minute := 59, [123].time.Second := 59, [123].time.DST_ON := 1, [124].log_data[0].min := 1.0, [124].log_data[0].max := 1.0, [124].log_data[0].total := 3600.0, [124].log_data[0].time := 3600.0, [124].log_data[0].valid := 1, [124].log_data[1].time := 3600.0, [124].log_data[1].valid := 1, [124].log_data[2].max := 1.0, [124].log_data[2].total := 435.75, [124].log_data[2].time := 3600.0, [124].log_data[2].maxminute := 52, [124].log_data[2].valid := 1, [124].log_data[3].time := 3600.0, [124].log_data[3].valid := 1,
        [124].log_data[4].min := 0.594375, [124].log_data[4].max := 1.0074999, [124].log_data[4].total := 2984.0364, [124].log_data[4].time := 3600.0, [124].log_data[4].maxminute := 52, [124].log_data[4].valid := 1, [124].log_data[5].max := 7.2275, [124].log_data[5].total := 3058.0574, [124].log_data[5].time := 3600.0, [124].log_data[5].maxminute := 55, [124].log_data[5].valid := 1, [124].log_data[6].valid := 1, [124].log_data[7].valid := 1, [124].log_data[8].valid := 1, [124].log_data[9].valid := 1, [124].log_data[10].valid := 1, [124].log_data[11].valid := 1, [124].log_data[12].valid := 1, [124].log_data[13].valid := 1, [124].log_data[14].valid := 1, [124].log_data[15].valid := 1, [124].log_data[16].valid := 1, [124].log_data[17].valid := 1, [124].log_data[18].valid := 1, [124].log_data[19].valid := 1, [124].time.Year := 2022, [124].time.Month := 5, [124].time.Day := 1, [124].time.Hour := 21, [124].time.Minute := 59, [124].time.Second := 59, [124].time.DST_ON := 1, [125].log_data[0].min := 1.0, [125].log_data[0].max := 1.0, [125].log_data[0].total := 3600.0, [125].log_data[0].time := 3600.0, [125].log_data[0].valid := 1, [125].log_data[1].time := 3600.0, [125].log_data[1].valid := 1, [125].log_data[2].max := 1.0, [125].log_data[2].total := 74.25, [125].log_data[2].time := 3600.0, [125].log_data[2].minminute := 1, [125].log_data[2].valid := 1, [125].log_data[3].time := 3600.0, [125].log_data[3].valid := 1, [125].log_data[4].min := 0.48749998, [125].log_data[4].max := 0.964375, [125].log_data[4].total := 2771.7322, [125].log_data[4].time := 3600.0, [125].log_data[4].minminute := 1, [125].log_data[4].maxminute := 57, [125].log_data[4].valid := 1, [125].log_data[5].max := 7.07125, [125].log_data[5].total := 564.2192, [125].log_data[5].time := 3600.0, [125].log_data[5].minminute := 1, [125].log_data[5].valid := 1, [125].log_data[6].valid := 1, [125].log_data[7].valid := 1,
        [125].log_data[8].valid := 1, [125].log_data[9].valid := 1, [125].log_data[10].valid := 1, [125].log_data[11].valid := 1, [125].log_data[12].valid := 1, [125].log_data[13].valid := 1, [125].log_data[14].valid := 1, [125].log_data[15].valid := 1, [125].log_data[16].valid := 1, [125].log_data[17].valid := 1, [125].log_data[18].valid := 1, [125].log_data[19].valid := 1, [125].time.Year := 2022, [125].time.Month := 5, [125].time.Day := 1, [125].time.Hour := 22, [125].time.Minute := 59, [125].time.Second := 59, [125].time.DST_ON := 1, [126].log_data[0].min := 1.0, [126].log_data[0].max := 1.0, [126].log_data[0].total := 3600.0, [126].log_data[0].time := 3600.0, [126].log_data[0].valid := 1, [126].log_data[1].max := 1.0, [126].log_data[1].total := 495.0, [126].log_data[1].time := 3600.0, [126].log_data[1].maxminute := 12, [126].log_data[1].valid := 1, [126].log_data[2].time := 3600.0, [126].log_data[2].valid := 1, [126].log_data[3].time := 3600.0, [126].log_data[3].valid := 1, [126].log_data[4].min := 0.48749998, [126].log_data[4].max := 1.00875, [126].log_data[4].total := 2602.8186, [126].log_data[4].time := 3600.0, [126].log_data[4].minminute := 21, [126].log_data[4].maxminute := 12, [126].log_data[4].valid := 1, [126].log_data[5].max := 7.1699996, [126].log_data[5].total := 3478.0938, [126].log_data[5].time := 3600.0, [126].log_data[5].maxminute := 13, [126].log_data[5].valid := 1, [126].log_data[6].valid := 1, [126].log_data[7].valid := 1, [126].log_data[8].valid := 1, [126].log_data[9].valid := 1, [126].log_data[10].valid := 1, [126].log_data[11].valid := 1, [126].log_data[12].valid := 1, [126].log_data[13].valid := 1, [126].log_data[14].valid := 1, [126].log_data[15].valid := 1, [126].log_data[16].valid := 1, [126].log_data[17].valid := 1, [126].log_data[18].valid := 1, [126].log_data[19].valid := 1, [126].time.Year := 2022,
        [126].time.Month := 5, [126].time.Day := 1, [126].time.Hour := 23, [126].time.Minute := 59, [126].time.Second := 59, [126].time.DST_ON := 1, [127].log_data[0].min := 1.0, [127].log_data[0].max := 1.0, [127].log_data[0].total := 3600.0, [127].log_data[0].time := 3600.0, [127].log_data[0].valid := 1, [127].log_data[1].time := 3600.0, [127].log_data[1].valid := 1, [127].log_data[2].time := 3600.0, [127].log_data[2].valid := 1, [127].log_data[3].time := 3600.0, [127].log_data[3].valid := 1, [127].log_data[4].min := 0.77937496, [127].log_data[4].max := 0.97937495, [127].log_data[4].total := 3256.1265, [127].log_data[4].time := 3600.0, [127].log_data[4].maxminute := 59, [127].log_data[4].valid := 1, [127].log_data[5].max := 0.0012500001, [127].log_data[5].total := 0.058437455, [127].log_data[5].time := 3600.0, [127].log_data[5].valid := 1, [127].log_data[6].valid := 1, [127].log_data[7].valid := 1, [127].log_data[8].valid := 1, [127].log_data[9].valid := 1, [127].log_data[10].valid := 1, [127].log_data[11].valid := 1, [127].log_data[12].valid := 1, [127].log_data[13].valid := 1, [127].log_data[14].valid := 1, [127].log_data[15].valid := 1, [127].log_data[16].valid := 1, [127].log_data[17].valid := 1, [127].log_data[18].valid := 1, [127].log_data[19].valid := 1, [127].time.Year := 2022, [127].time.Month := 5, [127].time.Day := 2, [127].time.Minute := 59, [127].time.Second := 59, [127].time.DST_ON := 1, [128].log_data[0].min := 1.0, [128].log_data[0].max := 1.0, [128].log_data[0].total := 3600.0, [128].log_data[0].time := 3600.0, [128].log_data[0].valid := 1, [128].log_data[1].time := 3600.0, [128].log_data[1].valid := 1, [128].log_data[2].max := 1.0, [128].log_data[2].total := 477.5, [128].log_data[2].time := 3600.0, [128].log_data[2].maxminute := 18, [128].log_data[2].valid := 1, [128].log_data[3].time := 3600.0,
        [128].log_data[3].valid := 1, [128].log_data[4].min := 0.48749998, [128].log_data[4].max := 1.003125, [128].log_data[4].total := 2606.4675, [128].log_data[4].time := 3600.0, [128].log_data[4].minminute := 26, [128].log_data[4].maxminute := 18, [128].log_data[4].valid := 1, [128].log_data[5].max := 7.2375, [128].log_data[5].total := 3394.9487, [128].log_data[5].time := 3600.0, [128].log_data[5].maxminute := 19, [128].log_data[5].valid := 1, [128].log_data[6].valid := 1, [128].log_data[7].valid := 1, [128].log_data[8].valid := 1, [128].log_data[9].valid := 1, [128].log_data[10].valid := 1, [128].log_data[11].valid := 1, [128].log_data[12].valid := 1, [128].log_data[13].valid := 1, [128].log_data[14].valid := 1, [128].log_data[15].valid := 1, [128].log_data[16].valid := 1, [128].log_data[17].valid := 1, [128].log_data[18].valid := 1, [128].log_data[19].valid := 1, [128].time.Year := 2022, [128].time.Month := 5, [128].time.Day := 2, [128].time.Hour := 1, [128].time.Minute := 59, [128].time.Second := 59, [128].time.DST_ON := 1, [129].log_data[0].min := 1.0, [129].log_data[0].max := 1.0, [129].log_data[0].total := 3599.999, [129].log_data[0].time := 3599.999, [129].log_data[0].valid := 1, [129].log_data[1].time := 3599.999, [129].log_data[1].valid := 1, [129].log_data[2].time := 3599.999, [129].log_data[2].valid := 1, [129].log_data[3].time := 3599.999, [129].log_data[3].valid := 1, [129].log_data[4].min := 0.625625, [129].log_data[4].max := 0.84124994, [129].log_data[4].total := 2682.6807, [129].log_data[4].time := 3599.999, [129].log_data[4].maxminute := 58, [129].log_data[4].valid := 1, [129].log_data[5].max := 0.0012500001, [129].log_data[5].total := 0.046874966, [129].log_data[5].time := 3599.999, [129].log_data[5].valid := 1, [129].log_data[6].valid := 1, [129].log_data[7].valid := 1, [129].log_data[8].valid := 1, [129].log_data[9].valid := 1, [129].log_data[10].valid := 1,
        [129].log_data[11].valid := 1, [129].log_data[12].valid := 1, [129].log_data[13].valid := 1, [129].log_data[14].valid := 1, [129].log_data[15].valid := 1, [129].log_data[16].valid := 1, [129].log_data[17].valid := 1, [129].log_data[18].valid := 1, [129].log_data[19].valid := 1, [129].time.Year := 2022, [129].time.Month := 5, [129].time.Day := 2, [129].time.Hour := 2, [129].time.Minute := 59, [129].time.Second := 59, [129].time.DST_ON := 1, [130].log_data[0].min := 1.0, [130].log_data[0].max := 1.0, [130].log_data[0].total := 3600.001, [130].log_data[0].time := 3600.001, [130].log_data[0].valid := 1, [130].log_data[1].time := 3600.001, [130].log_data[1].valid := 1, [130].log_data[2].time := 3600.001, [130].log_data[2].valid := 1, [130].log_data[3].time := 3600.001, [130].log_data[3].valid := 1, [130].log_data[4].min := 0.84062505, [130].log_data[4].max := 0.9024999, [130].log_data[4].total := 3164.4207, [130].log_data[4].time := 3600.001, [130].log_data[4].maxminute := 46, [130].log_data[4].valid := 1, [130].log_data[5].max := 0.0012500001, [130].log_data[5].total := 0.015937494, [130].log_data[5].time := 3600.001, [130].log_data[5].valid := 1, [130].log_data[6].valid := 1, [130].log_data[7].valid := 1, [130].log_data[8].valid := 1, [130].log_data[9].valid := 1, [130].log_data[10].valid := 1, [130].log_data[11].valid := 1, [130].log_data[12].valid := 1, [130].log_data[13].valid := 1, [130].log_data[14].valid := 1, [130].log_data[15].valid := 1, [130].log_data[16].valid := 1, [130].log_data[17].valid := 1, [130].log_data[18].valid := 1, [130].log_data[19].valid := 1, [130].time.Year := 2022, [130].time.Month := 5, [130].time.Day := 2, [130].time.Hour := 3, [130].time.Minute := 59, [130].time.Second := 59, [130].time.DST_ON := 1, [131].log_data[0].min := 1.0, [131].log_data[0].max := 1.0,
        [131].log_data[0].total := 3600.0, [131].log_data[0].time := 3600.0, [131].log_data[0].valid := 1, [131].log_data[1].time := 3600.0, [131].log_data[1].valid := 1, [131].log_data[2].time := 3600.0, [131].log_data[2].valid := 1, [131].log_data[3].time := 3600.0, [131].log_data[3].valid := 1, [131].log_data[4].min := 0.901875, [131].log_data[4].max := 0.94875, [131].log_data[4].total := 3349.2659, [131].log_data[4].time := 3600.0, [131].log_data[4].maxminute := 43, [131].log_data[4].valid := 1, [131].log_data[5].max := 0.0012500001, [131].log_data[5].total := 0.024374986, [131].log_data[5].time := 3600.0, [131].log_data[5].valid := 1, [131].log_data[6].valid := 1, [131].log_data[7].valid := 1, [131].log_data[8].valid := 1, [131].log_data[9].valid := 1, [131].log_data[10].valid := 1, [131].log_data[11].valid := 1, [131].log_data[12].valid := 1, [131].log_data[13].valid := 1, [131].log_data[14].valid := 1, [131].log_data[15].valid := 1, [131].log_data[16].valid := 1, [131].log_data[17].valid := 1, [131].log_data[18].valid := 1, [131].log_data[19].valid := 1, [131].time.Year := 2022, [131].time.Month := 5, [131].time.Day := 2, [131].time.Hour := 4, [131].time.Minute := 59, [131].time.Second := 59, [131].time.DST_ON := 1, [132].log_data[0].min := 1.0, [132].log_data[0].max := 1.0, [132].log_data[0].total := 3600.0, [132].log_data[0].time := 3600.0, [132].log_data[0].valid := 1, [132].log_data[1].time := 3600.0, [132].log_data[1].valid := 1, [132].log_data[2].time := 3600.0, [132].log_data[2].valid := 1, [132].log_data[3].time := 3600.0, [132].log_data[3].valid := 1, [132].log_data[4].min := 0.948125, [132].log_data[4].max := 0.97937495, [132].log_data[4].total := 3473.9204, [132].log_data[4].time := 3600.0, [132].log_data[4].maxminute := 44, [132].log_data[4].valid := 1, [132].log_data[5].max := 0.0012500001, [132].log_data[5].total := 0.036562476, [132].log_data[5].time := 3600.0,
        [132].log_data[5].valid := 1, [132].log_data[6].valid := 1, [132].log_data[7].valid := 1, [132].log_data[8].valid := 1, [132].log_data[9].valid := 1, [132].log_data[10].valid := 1, [132].log_data[11].valid := 1, [132].log_data[12].valid := 1, [132].log_data[13].valid := 1, [132].log_data[14].valid := 1, [132].log_data[15].valid := 1, [132].log_data[16].valid := 1, [132].log_data[17].valid := 1, [132].log_data[18].valid := 1, [132].log_data[19].valid := 1, [132].time.Year := 2022, [132].time.Month := 5, [132].time.Day := 2, [132].time.Hour := 5, [132].time.Minute := 59, [132].time.Second := 59, [132].time.DST_ON := 1, [133].log_data[0].min := 1.0, [133].log_data[0].max := 1.0, [133].log_data[0].total := 3600.0, [133].log_data[0].time := 3600.0, [133].log_data[0].valid := 1, [133].log_data[1].max := 1.0, [133].log_data[1].total := 472.0, [133].log_data[1].time := 3600.0, [133].log_data[1].maxminute := 40, [133].log_data[1].valid := 1, [133].log_data[2].time := 3600.0, [133].log_data[2].valid := 1, [133].log_data[3].time := 3600.0, [133].log_data[3].valid := 1, [133].log_data[4].min := 0.48749998, [133].log_data[4].max := 1.0068749, [133].log_data[4].total := 3143.3062, [133].log_data[4].time := 3600.0, [133].log_data[4].minminute := 49, [133].log_data[4].maxminute := 41, [133].log_data[4].valid := 1, [133].log_data[5].max := 7.1675005, [133].log_data[5].total := 3322.352, [133].log_data[5].time := 3600.0, [133].log_data[5].maxminute := 41, [133].log_data[5].valid := 1, [133].log_data[6].valid := 1, [133].log_data[7].valid := 1, [133].log_data[8].valid := 1, [133].log_data[9].valid := 1, [133].log_data[10].valid := 1, [133].log_data[11].valid := 1, [133].log_data[12].valid := 1, [133].log_data[13].valid := 1, [133].log_data[14].valid := 1, [133].log_data[15].valid := 1, [133].log_data[16].valid := 1, [133].log_data[17].valid := 1,
        [133].log_data[18].valid := 1, [133].log_data[19].valid := 1, [133].time.Year := 2022, [133].time.Month := 5, [133].time.Day := 2, [133].time.Hour := 6, [133].time.Minute := 59, [133].time.Second := 59, [133].time.DST_ON := 1, [134].log_data[0].min := 1.0, [134].log_data[0].max := 1.0, [134].log_data[0].total := 3600.0, [134].log_data[0].time := 3600.0, [134].log_data[0].valid := 1, [134].log_data[1].time := 3600.0, [134].log_data[1].valid := 1, [134].log_data[2].time := 3600.0, [134].log_data[2].valid := 1, [134].log_data[3].time := 3600.0, [134].log_data[3].valid := 1, [134].log_data[4].min := 0.50374997, [134].log_data[4].max := 0.71875, [134].log_data[4].total := 2085.5242, [134].log_data[4].time := 3600.0, [134].log_data[4].maxminute := 59, [134].log_data[4].valid := 1, [134].log_data[5].max := 0.0012500001, [134].log_data[5].total := 0.007812502, [134].log_data[5].time := 3600.0, [134].log_data[5].valid := 1, [134].log_data[6].valid := 1, [134].log_data[7].valid := 1, [134].log_data[8].valid := 1, [134].log_data[9].valid := 1, [134].log_data[10].valid := 1, [134].log_data[11].valid := 1, [134].log_data[12].valid := 1, [134].log_data[13].valid := 1, [134].log_data[14].valid := 1, [134].log_data[15].valid := 1, [134].log_data[16].valid := 1, [134].log_data[17].valid := 1, [134].log_data[18].valid := 1, [134].log_data[19].valid := 1, [134].time.Year := 2022, [134].time.Month := 5, [134].time.Day := 2, [134].time.Hour := 7, [134].time.Minute := 59, [134].time.Second := 59, [134].time.DST_ON := 1, [135].log_data[0].min := 1.0, [135].log_data[0].max := 1.0, [135].log_data[0].total := 3600.499, [135].log_data[0].time := 3600.499, [135].log_data[0].valid := 1, [135].log_data[1].time := 3600.499, [135].log_data[1].valid := 1, [135].log_data[2].max := 1.0, [135].log_data[2].total := 81.25,
        [135].log_data[2].time := 3600.499, [135].log_data[2].maxminute := 58, [135].log_data[2].valid := 1, [135].log_data[3].time := 3600.499, [135].log_data[3].valid := 1, [135].log_data[4].min := 0.71875, [135].log_data[4].max := 1.00625, [135].log_data[4].total := 3175.9656, [135].log_data[4].time := 3600.499, [135].log_data[4].maxminute := 58, [135].log_data[4].valid := 1, [135].log_data[5].max := 7.24625, [135].log_data[5].total := 525.23517, [135].log_data[5].time := 3600.499, [135].log_data[5].maxminute := 59, [135].log_data[5].valid := 1, [135].log_data[6].valid := 1, [135].log_data[7].valid := 1, [135].log_data[8].valid := 1, [135].log_data[9].valid := 1, [135].log_data[10].valid := 1, [135].log_data[11].valid := 1, [135].log_data[12].valid := 1, [135].log_data[13].valid := 1, [135].log_data[14].valid := 1, [135].log_data[15].valid := 1, [135].log_data[16].valid := 1, [135].log_data[17].valid := 1, [135].log_data[18].valid := 1, [135].log_data[19].valid := 1, [135].time.Year := 2022, [135].time.Month := 5, [135].time.Day := 2, [135].time.Hour := 8, [135].time.Minute := 59, [135].time.Second := 59, [135].time.DST_ON := 1, [136].log_data[0].min := 1.0, [136].log_data[0].max := 1.0, [136].log_data[0].total := 3600.0, [136].log_data[0].time := 3600.0, [136].log_data[0].valid := 1, [136].log_data[1].time := 3600.0, [136].log_data[1].valid := 1, [136].log_data[2].max := 1.0, [136].log_data[2].total := 416.25, [136].log_data[2].time := 3600.0, [136].log_data[2].minminute := 6, [136].log_data[2].valid := 1, [136].log_data[3].time := 3600.0, [136].log_data[3].valid := 1, [136].log_data[4].min := 0.48749998, [136].log_data[4].max := 0.964375, [136].log_data[4].total := 2683.7585, [136].log_data[4].time := 3600.0, [136].log_data[4].minminute := 7, [136].log_data[4].valid := 1, [136].log_data[5].max := 7.2525, [136].log_data[5].total := 3013.844, [136].log_data[5].time := 3600.0,
